LIN {X 0,Y 508.464,Z 856.949,A -85,B 0,C 180,E1 23996.123,E2 23996.123} C_VEL
LIN {X 0,Y 510.353,Z 835.895,A -85,B 0,C 180,E1 23994.699,E2 23994.699} C_VEL
LIN {X 0,Y 512.126,Z 815.37,A -85,B 0,C 180,E1 23993.529,E2 23993.529} C_VEL
LIN {X 0,Y 513.642,Z 794.189,A -85,B 0,C 180,E1 23992.545,E2 23992.545} C_VEL
LIN {X 0,Y 515.036,Z 772.161,A -85,B 0,C 180,E1 23991.717,E2 23991.717} C_VEL
LIN {X 0,Y 516.1,Z 749.861,A -85,B 0,C 180,E1 23991.103,E2 23991.103} C_VEL
LIN {X 0,Y 516.88,Z 725.33,A -85,B 0,C 180,E1 23990.627,E2 23990.627} C_VEL
LIN {X 0,Y 520.489,Z 517.525,A -85,B 0,C 180,E1 23987.247,E2 23987.247} C_VEL
LIN {X 0,Y 522.256,Z 415.583,A -85,B 0,C 180,E1 23985.539,E2 23985.539} C_VEL
LIN {X 0,Y 521.351,Z 412.142,A -85,B 0,C 180,E1 23985.377,E2 23985.377} C_VEL
LIN {X 0,Y 506.153,Z 388.849,A -85,B 0,C 180,E1 23983.194,E2 23983.194} C_VEL
LIN {X 0,Y 500.353,Z 377.109,A -85,B 0,C 180,E1 23981.409,E2 23981.409} C_VEL
LIN {X 0,Y 498.571,Z 373.357,A -85,B 0,C 180,E1 23980.826,E2 23980.826} C_VEL
LIN {X 0,Y 496.991,Z 370.279,A -85,B 0,C 180,E1 23980.325,E2 23980.325} C_VEL
LIN {X 0,Y 496.775,Z 369.171,A -85,B 0,C 180,E1 23980.17,E2 23980.17} C_VEL
LIN {X 0,Y 496.727,Z 369.173,A -85,B 0,C 180,E1 23976.714,E2 23976.714} C_VEL
LIN {X 0,Y 496.716,Z 369.158,A -85,B 0,C 180,E1 23973.146,E2 23973.146} C_VEL
LIN {X 0,Y 496.773,Z 369.141,A -85,B 0,C 180,E1 23969.81,E2 23969.81} C_VEL
LIN {X 0,Y 496.717,Z 369.17,A -85,B 0,C 180,E1 23966.409,E2 23966.409} C_VEL
LIN {X 0,Y 496.704,Z 369.151,A -85,B 0,C 180,E1 23962.861,E2 23962.861} C_VEL
LIN {X 0,Y 496.76,Z 369.159,A -85,B 0,C 180,E1 23959.519,E2 23959.519} C_VEL
LIN {X 0,Y 496.704,Z 369.158,A -85,B 0,C 180,E1 23956.128,E2 23956.128} C_VEL
LIN {X 0,Y 496.693,Z 369.168,A -85,B 0,C 180,E1 23952.556,E2 23952.556} C_VEL
LIN {X 0,Y 496.742,Z 369.166,A -85,B 0,C 180,E1 23949.149,E2 23949.149} C_VEL
LIN {X 0,Y 496.691,Z 369.172,A -85,B 0,C 180,E1 23945.892,E2 23945.892} C_VEL
LIN {X 0,Y 496.69,Z 369.167,A -85,B 0,C 180,E1 23942.307,E2 23942.307} C_VEL
LIN {X 0,Y 496.758,Z 369.164,A -85,B 0,C 180,E1 23938.962,E2 23938.962} C_VEL
LIN {X 0,Y 496.711,Z 369.174,A -85,B 0,C 180,E1 23935.497,E2 23935.497} C_VEL
LIN {X 0,Y 496.703,Z 369.171,A -85,B 0,C 180,E1 23932.002,E2 23932.002} C_VEL
LIN {X 0,Y 496.76,Z 369.165,A -85,B 0,C 180,E1 23928.624,E2 23928.624} C_VEL
LIN {X 0,Y 496.725,Z 369.174,A -85,B 0,C 180,E1 23925.188,E2 23925.188} C_VEL
LIN {X 0,Y 496.712,Z 369.149,A -85,B 0,C 180,E1 23921.698,E2 23921.698} C_VEL
LIN {X 0,Y 496.768,Z 369.16,A -85,B 0,C 180,E1 23918.263,E2 23918.263} C_VEL
LIN {X 0,Y 496.746,Z 369.154,A -85,B 0,C 180,E1 23914.74,E2 23914.74} C_VEL
LIN {X 0,Y 496.721,Z 369.154,A -85,B 0,C 180,E1 23911.243,E2 23911.243} C_VEL
LIN {X 0,Y 496.754,Z 369.169,A -85,B 0,C 180,E1 23907.765,E2 23907.765} C_VEL
LIN {X 0,Y 496.766,Z 369.148,A -85,B 0,C 180,E1 23904.289,E2 23904.289} C_VEL
LIN {X 0,Y 496.733,Z 369.148,A -85,B 0,C 180,E1 23900.792,E2 23900.792} C_VEL
LIN {X 0,Y 496.803,Z 369.408,A -85,B 0,C 180,E1 23897.786,E2 23897.786} C_VEL
LIN {X 0,Y 498.038,Z 372.602,A -85,B 0,C 180,E1 23897.561,E2 23897.561} C_VEL
LIN {X 0,Y 500.713,Z 375.613,A -85,B 0,C 180,E1 23897.161,E2 23897.161} C_VEL
LIN {X 0,Y 503.415,Z 379.529,A -85,B 0,C 180,E1 23896.747,E2 23896.747} C_VEL
LIN {X 0,Y 505.239,Z 382.053,A -85,B 0,C 180,E1 23896.474,E2 23896.474} C_VEL
LIN {X 0,Y 515.597,Z 396.493,A -85,B 0,C 180,E1 23894.982,E2 23894.982} C_VEL
LIN {X 0,Y 522.157,Z 406.331,A -85,B 0,C 180,E1 23894.073,E2 23894.073} C_VEL
LIN {X 0,Y 521.852,Z 421.709,A -85,B 0,C 180,E1 23893.817,E2 23893.817} C_VEL
LIN {X 0,Y 520.999,Z 429.411,A -85,B 0,C 180,E1 23893.763,E2 23893.763} C_VEL
LIN {X 0,Y 516.075,Z 450.049,A -85,B 0,C 180,E1 23893.901,E2 23893.901} C_VEL
LIN {X 0,Y 515.405,Z 456.658,A -85,B 0,C 180,E1 23893.847,E2 23893.847} C_VEL
LIN {X 0,Y 511.252,Z 667.268,A -85,B 0,C 180,E1 23890.36,E2 23890.36} C_VEL
LIN {X 0,Y 510.217,Z 713.646,A -85,B 0,C 180,E1 23889.568,E2 23889.568} C_VEL
LIN {X 0,Y 509.142,Z 735.14,A -85,B 0,C 180,E1 23889.014,E2 23889.014} C_VEL
LIN {X 0,Y 507.831,Z 756.494,A -85,B 0,C 180,E1 23888.289,E2 23888.289} C_VEL
LIN {X 0,Y 506.068,Z 778.939,A -85,B 0,C 180,E1 23887.296,E2 23887.296} C_VEL
LIN {X 0,Y 504.16,Z 801.229,A -85,B 0,C 180,E1 23886.082,E2 23886.082} C_VEL
LIN {X 0,Y 502.303,Z 820.309,A -85,B 0,C 180,E1 23884.835,E2 23884.835} C_VEL
LIN {X 0,Y 500.115,Z 841.41,A -85,B 0,C 180,E1 23883.211,E2 23883.211} C_VEL
LIN {X 0,Y 498.19,Z 859.526,A -85,B 0,C 180,E1 23881.585,E2 23881.585} C_VEL
LIN {X 0,Y 496.137,Z 878.107,A -85,B 0,C 180,E1 23879.649,E2 23879.649} C_VEL
LIN {X 0,Y 494.326,Z 895.329,A -85,B 0,C 180,E1 23877.589,E2 23877.589} C_VEL
LIN {X 0,Y 492.667,Z 911.402,A -85,B 0,C 180,E1 23875.351,E2 23875.351} C_VEL
LIN {X 0,Y 491.199,Z 926.819,A -85,B 0,C 180,E1 23872.876,E2 23872.876} C_VEL
LIN {X 0,Y 490.091,Z 940.046,A -85,B 0,C 180,E1 23870.415,E2 23870.415} C_VEL
LIN {X 0,Y 489.24,Z 951.697,A -85,B 0,C 180,E1 23867.849,E2 23867.849} C_VEL
LIN {X 0,Y 488.644,Z 961.975,A -85,B 0,C 180,E1 23865.181,E2 23865.181} C_VEL
LIN {X 0,Y 488.286,Z 969.634,A -85,B 0,C 180,E1 23862.775,E2 23862.775} C_VEL
LIN {X 0,Y 488.034,Z 976.716,A -85,B 0,C 180,E1 23860.027,E2 23860.027} C_VEL
LIN {X 0,Y 487.954,Z 981.385,A -85,B 0,C 180,E1 23857.653,E2 23857.653} C_VEL
LIN {X 0,Y 487.914,Z 985.231,A -85,B 0,C 180,E1 23854.937,E2 23854.937} C_VEL
LIN {X 0,Y 487.909,Z 987.232,A -85,B 0,C 180,E1 23852.466,E2 23852.466} C_VEL
LIN {X 0,Y 487.908,Z 987.992,A -85,B 0,C 180,E1 23849.882,E2 23849.882} C_VEL
LIN {X 0,Y 487.904,Z 987.148,A -85,B 0,C 180,E1 23847.298,E2 23847.298} C_VEL
LIN {X 0,Y 487.918,Z 984.97,A -85,B 0,C 180,E1 23844.709,E2 23844.709} C_VEL
LIN {X 0,Y 487.969,Z 981.128,A -85,B 0,C 180,E1 23842.11,E2 23842.11} C_VEL
LIN {X 0,Y 488.079,Z 975.882,A -85,B 0,C 180,E1 23839.496,E2 23839.496} C_VEL
LIN {X 0,Y 488.32,Z 968.838,A -85,B 0,C 180,E1 23836.864,E2 23836.864} C_VEL
LIN {X 0,Y 488.735,Z 960.16,A -85,B 0,C 180,E1 23834.213,E2 23834.213} C_VEL
LIN {X 0,Y 489.315,Z 950.523,A -85,B 0,C 180,E1 23831.784,E2 23831.784} C_VEL
LIN {X 0,Y 490.256,Z 937.895,A -85,B 0,C 180,E1 23829.079,E2 23829.079} C_VEL
LIN {X 0,Y 491.348,Z 925.2,A -85,B 0,C 180,E1 23826.75,E2 23826.75} C_VEL
LIN {X 0,Y 492.769,Z 910.298,A -85,B 0,C 180,E1 23824.396,E2 23824.396} C_VEL
LIN {X 0,Y 494.415,Z 894.536,A -85,B 0,C 180,E1 23822.219,E2 23822.219} C_VEL
LIN {X 0,Y 496.191,Z 877.593,A -85,B 0,C 180,E1 23820.203,E2 23820.203} C_VEL
LIN {X 0,Y 498.305,Z 858.41,A -85,B 0,C 180,E1 23818.22,E2 23818.22} C_VEL
LIN {X 0,Y 500.249,Z 840.17,A -85,B 0,C 180,E1 23816.593,E2 23816.593} C_VEL
LIN {X 0,Y 502.368,Z 819.664,A -85,B 0,C 180,E1 23815.03,E2 23815.03} C_VEL
LIN {X 0,Y 504.234,Z 800.49,A -85,B 0,C 180,E1 23813.783,E2 23813.783} C_VEL
LIN {X 0,Y 506.062,Z 779,A -85,B 0,C 180,E1 23812.617,E2 23812.617} C_VEL
LIN {X 0,Y 507.824,Z 756.603,A -85,B 0,C 180,E1 23811.625,E2 23811.625} C_VEL
LIN {X 0,Y 509.13,Z 735.348,A -85,B 0,C 180,E1 23810.903,E2 23810.903} C_VEL
LIN {X 0,Y 510.191,Z 714.187,A -85,B 0,C 180,E1 23810.354,E2 23810.354} C_VEL
LIN {X 0,Y 511.145,Z 673.08,A -85,B 0,C 180,E1 23809.645,E2 23809.645} C_VEL
LIN {X 0,Y 515.353,Z 459.338,A -85,B 0,C 180,E1 23806.108,E2 23806.108} C_VEL
LIN {X 0,Y 516.278,Z 409.582,A -85,B 0,C 180,E1 23805.257,E2 23805.257} C_VEL
LIN {X 0,Y 502.991,Z 390.592,A -85,B 0,C 180,E1 23803.338,E2 23803.338} C_VEL
LIN {X 0,Y 498.896,Z 385.123,A -85,B 0,C 180,E1 23802.719,E2 23802.719} C_VEL
LIN {X 0,Y 495.764,Z 380.744,A -85,B 0,C 180,E1 23802.23,E2 23802.23} C_VEL
LIN {X 0,Y 493.031,Z 376.923,A -85,B 0,C 180,E1 23801.793,E2 23801.793} C_VEL
LIN {X 0,Y 492.228,Z 375.754,A -85,B 0,C 180,E1 23801.663,E2 23801.663} C_VEL
LIN {X 0,Y 489.757,Z 373.065,A -85,B 0,C 180,E1 23801.275,E2 23801.275} C_VEL
LIN {X 0,Y 488.804,Z 370.162,A -85,B 0,C 180,E1 23801.073,E2 23801.073} C_VEL
LIN {X 0,Y 488.818,Z 370.152,A -85,B 0,C 180,E1 23797.481,E2 23797.481} C_VEL
LIN {X 0,Y 488.831,Z 370.129,A -85,B 0,C 180,E1 23793.866,E2 23793.866} C_VEL
LIN {X 0,Y 488.803,Z 370.14,A -85,B 0,C 180,E1 23790.332,E2 23790.332} C_VEL
LIN {X 0,Y 488.79,Z 370.162,A -85,B 0,C 180,E1 23786.746,E2 23786.746} C_VEL
LIN {X 0,Y 488.816,Z 370.127,A -85,B 0,C 180,E1 23783.252,E2 23783.252} C_VEL
LIN {X 0,Y 488.82,Z 370.159,A -85,B 0,C 180,E1 23779.725,E2 23779.725} C_VEL
LIN {X 0,Y 488.773,Z 370.134,A -85,B 0,C 180,E1 23776.276,E2 23776.276} C_VEL
LIN {X 0,Y 488.791,Z 370.156,A -85,B 0,C 180,E1 23772.763,E2 23772.763} C_VEL
LIN {X 0,Y 488.823,Z 370.157,A -85,B 0,C 180,E1 23769.299,E2 23769.299} C_VEL
LIN {X 0,Y 488.768,Z 370.161,A -85,B 0,C 180,E1 23765.871,E2 23765.871} C_VEL
LIN {X 0,Y 488.764,Z 370.161,A -85,B 0,C 180,E1 23762.228,E2 23762.228} C_VEL
LIN {X 0,Y 488.817,Z 370.159,A -85,B 0,C 180,E1 23758.828,E2 23758.828} C_VEL
LIN {X 0,Y 488.771,Z 370.163,A -85,B 0,C 180,E1 23755.307,E2 23755.307} C_VEL
LIN {X 0,Y 488.748,Z 370.163,A -85,B 0,C 180,E1 23751.885,E2 23751.885} C_VEL
LIN {X 0,Y 488.798,Z 370.16,A -85,B 0,C 180,E1 23748.436,E2 23748.436} C_VEL
LIN {X 0,Y 488.77,Z 370.165,A -85,B 0,C 180,E1 23745.064,E2 23745.064} C_VEL
LIN {X 0,Y 488.757,Z 370.14,A -85,B 0,C 180,E1 23741.514,E2 23741.514} C_VEL
LIN {X 0,Y 488.796,Z 370.152,A -85,B 0,C 180,E1 23738.017,E2 23738.017} C_VEL
LIN {X 0,Y 488.802,Z 370.15,A -85,B 0,C 180,E1 23734.561,E2 23734.561} C_VEL
LIN {X 0,Y 488.768,Z 370.137,A -85,B 0,C 180,E1 23731.098,E2 23731.098} C_VEL
LIN {X 0,Y 488.795,Z 370.155,A -85,B 0,C 180,E1 23727.593,E2 23727.593} C_VEL
LIN {X 0,Y 488.829,Z 370.157,A -85,B 0,C 180,E1 23724.054,E2 23724.054} C_VEL
LIN {X 0,Y 488.799,Z 370.271,A -85,B 0,C 180,E1 23720.776,E2 23720.776} C_VEL
LIN {X 0,Y 490.062,Z 373.556,A -85,B 0,C 180,E1 23720.273,E2 23720.273} C_VEL
LIN {X 0,Y 491.239,Z 375.449,A -85,B 0,C 180,E1 23719.927,E2 23719.927} C_VEL
LIN {X 0,Y 497.884,Z 388.868,A -85,B 0,C 180,E1 23717.812,E2 23717.812} C_VEL
LIN {X 0,Y 511.426,Z 409.267,A -85,B 0,C 180,E1 23715.777,E2 23715.777} C_VEL
LIN {X 0,Y 516.558,Z 417.775,A -85,B 0,C 180,E1 23715.037,E2 23715.037} C_VEL
LIN {X 0,Y 513.166,Z 591.207,A -85,B 0,C 180,E1 23712.135,E2 23712.135} C_VEL
LIN {X 0,Y 510.26,Z 740.048,A -85,B 0,C 180,E1 23709.677,E2 23709.677} C_VEL
LIN {X 0,Y 509.209,Z 762.982,A -85,B 0,C 180,E1 23709.115,E2 23709.115} C_VEL
LIN {X 0,Y 508.022,Z 782.983,A -85,B 0,C 180,E1 23708.457,E2 23708.457} C_VEL
LIN {X 0,Y 506.378,Z 805.177,A -85,B 0,C 180,E1 23707.523,E2 23707.523} C_VEL
LIN {X 0,Y 504.581,Z 826.539,A -85,B 0,C 180,E1 23706.407,E2 23706.407} C_VEL
LIN {X 0,Y 502.609,Z 847.281,A -85,B 0,C 180,E1 23705.09,E2 23705.09} C_VEL
LIN {X 0,Y 500.556,Z 867.467,A -85,B 0,C 180,E1 23703.59,E2 23703.59} C_VEL
LIN {X 0,Y 498.488,Z 886.631,A -85,B 0,C 180,E1 23701.902,E2 23701.902} C_VEL
LIN {X 0,Y 496.409,Z 905.703,A -85,B 0,C 180,E1 23699.965,E2 23699.965} C_VEL
LIN {X 0,Y 494.669,Z 921.952,A -85,B 0,C 180,E1 23698.055,E2 23698.055} C_VEL
LIN {X 0,Y 492.895,Z 938.97,A -85,B 0,C 180,E1 23695.754,E2 23695.754} C_VEL
LIN {X 0,Y 491.484,Z 953.859,A -85,B 0,C 180,E1 23693.438,E2 23693.438} C_VEL
LIN {X 0,Y 490.319,Z 967.096,A -85,B 0,C 180,E1 23691.03,E2 23691.03} C_VEL
LIN {X 0,Y 489.404,Z 979.297,A -85,B 0,C 180,E1 23688.46,E2 23688.46} C_VEL
LIN {X 0,Y 488.783,Z 989.073,A -85,B 0,C 180,E1 23686.029,E2 23686.029} C_VEL
LIN {X 0,Y 488.338,Z 998.352,A -85,B 0,C 180,E1 23683.256,E2 23683.256} C_VEL
LIN {X 0,Y 488.1,Z 1004.868,A -85,B 0,C 180,E1 23680.862,E2 23680.862} C_VEL
LIN {X 0,Y 487.978,Z 1010.636,A -85,B 0,C 180,E1 23678.127,E2 23678.127} C_VEL
LIN {X 0,Y 487.913,Z 1014.438,A -85,B 0,C 180,E1 23675.645,E2 23675.645} C_VEL
LIN {X 0,Y 487.89,Z 1016.986,A -85,B 0,C 180,E1 23672.937,E2 23672.937} C_VEL
LIN {X 0,Y 487.885,Z 1017.895,A -85,B 0,C 180,E1 23670.587,E2 23670.587} C_VEL
LIN {X 0,Y 487.914,Z 1017.393,A -85,B 0,C 180,E1 23667.769,E2 23667.769} C_VEL
LIN {X 0,Y 487.906,Z 1015.502,A -85,B 0,C 180,E1 23665.299,E2 23665.299} C_VEL
LIN {X 0,Y 487.933,Z 1011.876,A -85,B 0,C 180,E1 23662.584,E2 23662.584} C_VEL
LIN {X 0,Y 488.017,Z 1007.347,A -85,B 0,C 180,E1 23660.222,E2 23660.222} C_VEL
LIN {X 0,Y 488.242,Z 1000.825,A -85,B 0,C 180,E1 23657.585,E2 23657.585} C_VEL
LIN {X 0,Y 488.592,Z 992.944,A -85,B 0,C 180,E1 23655.06,E2 23655.06} C_VEL
LIN {X 0,Y 489.199,Z 982.338,A -85,B 0,C 180,E1 23652.257,E2 23652.257} C_VEL
LIN {X 0,Y 489.978,Z 971.429,A -85,B 0,C 180,E1 23649.829,E2 23649.829} C_VEL
LIN {X 0,Y 491.056,Z 958.469,A -85,B 0,C 180,E1 23647.37,E2 23647.37} C_VEL
LIN {X 0,Y 492.405,Z 944.233,A -85,B 0,C 180,E1 23645.02,E2 23645.02} C_VEL
LIN {X 0,Y 493.963,Z 928.434,A -85,B 0,C 180,E1 23642.78,E2 23642.78} C_VEL
LIN {X 0,Y 495.925,Z 910.148,A -85,B 0,C 180,E1 23640.536,E2 23640.536} C_VEL
LIN {X 0,Y 497.859,Z 892.56,A -85,B 0,C 180,E1 23638.662,E2 23638.662} C_VEL
LIN {X 0,Y 499.911,Z 873.362,A -85,B 0,C 180,E1 23636.91,E2 23636.91} C_VEL
LIN {X 0,Y 501.985,Z 853.573,A -85,B 0,C 180,E1 23635.347,E2 23635.347} C_VEL
LIN {X 0,Y 503.895,Z 833.882,A -85,B 0,C 180,E1 23634.037,E2 23634.037} C_VEL
LIN {X 0,Y 505.798,Z 812.769,A -85,B 0,C 180,E1 23632.848,E2 23632.848} C_VEL
LIN {X 0,Y 507.33,Z 792.54,A -85,B 0,C 180,E1 23631.918,E2 23631.918} C_VEL
LIN {X 0,Y 508.864,Z 769.286,A -85,B 0,C 180,E1 23631.071,E2 23631.071} C_VEL
LIN {X 0,Y 509.898,Z 748.81,A -85,B 0,C 180,E1 23630.516,E2 23630.516} C_VEL
LIN {X 0,Y 510.736,Z 722.059,A -85,B 0,C 180,E1 23630.006,E2 23630.006} C_VEL
LIN {X 0,Y 514.648,Z 514.981,A -85,B 0,C 180,E1 23626.601,E2 23626.601} C_VEL
LIN {X 0,Y 516.488,Z 417.402,A -85,B 0,C 180,E1 23624.948,E2 23624.948} C_VEL
LIN {X 0,Y 502.74,Z 395.952,A -85,B 0,C 180,E1 23622.935,E2 23622.935} C_VEL
LIN {X 0,Y 497.647,Z 388.466,A -85,B 0,C 180,E1 23622.149,E2 23622.149} C_VEL
LIN {X 0,Y 492.504,Z 378.211,A -85,B 0,C 180,E1 23620.515,E2 23620.515} C_VEL
LIN {X 0,Y 490.79,Z 374.486,A -85,B 0,C 180,E1 23619.921,E2 23619.921} C_VEL
LIN {X 0,Y 488.97,Z 371.128,A -85,B 0,C 180,E1 23619.338,E2 23619.338} C_VEL
LIN {X 0,Y 488.783,Z 370.16,A -85,B 0,C 180,E1 23619.178,E2 23619.178} C_VEL
LIN {X 0,Y 488.811,Z 370.153,A -85,B 0,C 180,E1 23615.659,E2 23615.659} C_VEL
LIN {X 0,Y 488.82,Z 370.155,A -85,B 0,C 180,E1 23612.128,E2 23612.128} C_VEL
LIN {X 0,Y 488.769,Z 370.135,A -85,B 0,C 180,E1 23608.733,E2 23608.733} C_VEL
LIN {X 0,Y 488.783,Z 370.145,A -85,B 0,C 180,E1 23605.181,E2 23605.181} C_VEL
LIN {X 0,Y 488.825,Z 370.146,A -85,B 0,C 180,E1 23601.729,E2 23601.729} C_VEL
LIN {X 0,Y 488.763,Z 370.135,A -85,B 0,C 180,E1 23598.239,E2 23598.239} C_VEL
LIN {X 0,Y 488.758,Z 370.164,A -85,B 0,C 180,E1 23594.647,E2 23594.647} C_VEL
LIN {X 0,Y 488.806,Z 370.162,A -85,B 0,C 180,E1 23591.205,E2 23591.205} C_VEL
LIN {X 0,Y 488.766,Z 370.162,A -85,B 0,C 180,E1 23587.759,E2 23587.759} C_VEL
LIN {X 0,Y 488.748,Z 370.164,A -85,B 0,C 180,E1 23584.223,E2 23584.223} C_VEL
LIN {X 0,Y 488.796,Z 370.162,A -85,B 0,C 180,E1 23580.82,E2 23580.82} C_VEL
LIN {X 0,Y 488.778,Z 370.157,A -85,B 0,C 180,E1 23577.42,E2 23577.42} C_VEL
LIN {X 0,Y 488.759,Z 370.16,A -85,B 0,C 180,E1 23573.893,E2 23573.893} C_VEL
LIN {X 0,Y 488.8,Z 370.158,A -85,B 0,C 180,E1 23570.463,E2 23570.463} C_VEL
LIN {X 0,Y 488.804,Z 370.154,A -85,B 0,C 180,E1 23566.996,E2 23566.996} C_VEL
LIN {X 0,Y 488.77,Z 370.141,A -85,B 0,C 180,E1 23563.597,E2 23563.597} C_VEL
LIN {X 0,Y 488.807,Z 370.159,A -85,B 0,C 180,E1 23560.15,E2 23560.15} C_VEL
LIN {X 0,Y 488.816,Z 370.128,A -85,B 0,C 180,E1 23556.679,E2 23556.679} C_VEL
LIN {X 0,Y 488.786,Z 370.162,A -85,B 0,C 180,E1 23553.123,E2 23553.123} C_VEL
LIN {X 0,Y 488.793,Z 370.139,A -85,B 0,C 180,E1 23549.516,E2 23549.516} C_VEL
LIN {X 0,Y 488.831,Z 370.133,A -85,B 0,C 180,E1 23546.055,E2 23546.055} C_VEL
LIN {X 0,Y 488.818,Z 370.155,A -85,B 0,C 180,E1 23542.443,E2 23542.443} C_VEL
LIN {X 0,Y 488.797,Z 370.162,A -85,B 0,C 180,E1 23538.896,E2 23538.896} C_VEL
LIN {X 0,Y 488.832,Z 370.403,A -85,B 0,C 180,E1 23538.816,E2 23538.816} C_VEL
LIN {X 0,Y 490.061,Z 373.569,A -85,B 0,C 180,E1 23538.581,E2 23538.581} C_VEL
LIN {X 0,Y 492.913,Z 376.68,A -85,B 0,C 180,E1 23538.136,E2 23538.136} C_VEL
LIN {X 0,Y 495.559,Z 380.548,A -85,B 0,C 180,E1 23537.71,E2 23537.71} C_VEL
LIN {X 0,Y 497.277,Z 382.868,A -85,B 0,C 180,E1 23537.442,E2 23537.442} C_VEL
LIN {X 0,Y 504.541,Z 392.801,A -85,B 0,C 180,E1 23536.339,E2 23536.339} C_VEL
LIN {X 0,Y 516.37,Z 409.728,A -85,B 0,C 180,E1 23534.64,E2 23534.64} C_VEL
LIN {X 0,Y 515.405,Z 456.658,A -85,B 0,C 180,E1 23533.847,E2 23533.847} C_VEL
LIN {X 0,Y 514.529,Z 464.362,A -85,B 0,C 180,E1 23533.795,E2 23533.795} C_VEL
LIN {X 0,Y 509.557,Z 484.99,A -85,B 0,C 180,E1 23533.94,E2 23533.94} C_VEL
LIN {X 0,Y 508.893,Z 491.597,A -85,B 0,C 180,E1 23533.886,E2 23533.886} C_VEL
LIN {X 0,Y 504.452,Z 702.056,A -85,B 0,C 180,E1 23530.374,E2 23530.374} C_VEL
LIN {X 0,Y 503.552,Z 723.847,A -85,B 0,C 180,E1 23529.915,E2 23529.915} C_VEL
LIN {X 0,Y 502.14,Z 747.778,A -85,B 0,C 180,E1 23529.189,E2 23529.189} C_VEL
LIN {X 0,Y 500.66,Z 767.864,A -85,B 0,C 180,E1 23528.39,E2 23528.39} C_VEL
LIN {X 0,Y 498.747,Z 789.324,A -85,B 0,C 180,E1 23527.327,E2 23527.327} C_VEL
LIN {X 0,Y 496.745,Z 809.274,A -85,B 0,C 180,E1 23526.134,E2 23526.134} C_VEL
LIN {X 0,Y 494.552,Z 829.67,A -85,B 0,C 180,E1 23524.684,E2 23524.684} C_VEL
LIN {X 0,Y 492.413,Z 848.758,A -85,B 0,C 180,E1 23523.103,E2 23523.103} C_VEL
LIN {X 0,Y 490.161,Z 867.608,A -85,B 0,C 180,E1 23521.273,E2 23521.273} C_VEL
LIN {X 0,Y 488.127,Z 885.24,A -85,B 0,C 180,E1 23519.307,E2 23519.307} C_VEL
LIN {X 0,Y 486.237,Z 901.358,A -85,B 0,C 180,E1 23517.224,E2 23517.224} C_VEL
LIN {X 0,Y 484.434,Z 917.974,A -85,B 0,C 180,E1 23514.749,E2 23514.749} C_VEL
LIN {X 0,Y 483.042,Z 932.215,A -85,B 0,C 180,E1 23512.293,E2 23512.293} C_VEL
LIN {X 0,Y 481.928,Z 944.678,A -85,B 0,C 180,E1 23509.763,E2 23509.763} C_VEL
LIN {X 0,Y 481.074,Z 956.154,A -85,B 0,C 180,E1 23507.038,E2 23507.038} C_VEL
LIN {X 0,Y 480.559,Z 964.819,A -85,B 0,C 180,E1 23504.579,E2 23504.579} C_VEL
LIN {X 0,Y 480.195,Z 972.938,A -85,B 0,C 180,E1 23501.772,E2 23501.772} C_VEL
LIN {X 0,Y 480.019,Z 978.499,A -85,B 0,C 180,E1 23499.349,E2 23499.349} C_VEL
LIN {X 0,Y 479.936,Z 983.262,A -85,B 0,C 180,E1 23496.578,E2 23496.578} C_VEL
LIN {X 0,Y 479.913,Z 986.027,A -85,B 0,C 180,E1 23494.181,E2 23494.181} C_VEL
LIN {X 0,Y 479.908,Z 987.75,A -85,B 0,C 180,E1 23491.313,E2 23491.313} C_VEL
LIN {X 0,Y 479.892,Z 987.813,A -85,B 0,C 180,E1 23488.925,E2 23488.925} C_VEL
LIN {X 0,Y 479.899,Z 986.563,A -85,B 0,C 180,E1 23486.297,E2 23486.297} C_VEL
LIN {X 0,Y 479.934,Z 983.86,A -85,B 0,C 180,E1 23483.781,E2 23483.781} C_VEL
LIN {X 0,Y 480.003,Z 979.68,A -85,B 0,C 180,E1 23481.134,E2 23481.134} C_VEL
LIN {X 0,Y 480.148,Z 973.768,A -85,B 0,C 180,E1 23478.469,E2 23478.469} C_VEL
LIN {X 0,Y 480.462,Z 966.602,A -85,B 0,C 180,E1 23475.875,E2 23475.875} C_VEL
LIN {X 0,Y 480.95,Z 957.861,A -85,B 0,C 180,E1 23473.33,E2 23473.33} C_VEL
LIN {X 0,Y 481.708,Z 947.373,A -85,B 0,C 180,E1 23470.731,E2 23470.731} C_VEL
LIN {X 0,Y 482.711,Z 935.413,A -85,B 0,C 180,E1 23468.239,E2 23468.239} C_VEL
LIN {X 0,Y 484.15,Z 920.709,A -85,B 0,C 180,E1 23465.607,E2 23465.607} C_VEL
LIN {X 0,Y 485.736,Z 906.057,A -85,B 0,C 180,E1 23463.34,E2 23463.34} C_VEL
LIN {X 0,Y 487.531,Z 889.966,A -85,B 0,C 180,E1 23461.19,E2 23461.19} C_VEL
LIN {X 0,Y 489.606,Z 872.681,A -85,B 0,C 180,E1 23459.167,E2 23459.167} C_VEL
LIN {X 0,Y 491.702,Z 854.474,A -85,B 0,C 180,E1 23457.337,E2 23457.337} C_VEL
LIN {X 0,Y 494.091,Z 833.949,A -85,B 0,C 180,E1 23455.56,E2 23455.56} C_VEL
LIN {X 0,Y 496.132,Z 815.146,A -85,B 0,C 180,E1 23454.17,E2 23454.17} C_VEL
LIN {X 0,Y 498.35,Z 793.207,A -85,B 0,C 180,E1 23452.799,E2 23452.799} C_VEL
LIN {X 0,Y 500.3,Z 772.386,A -85,B 0,C 180,E1 23451.722,E2 23451.722} C_VEL
LIN {X 0,Y 501.962,Z 750.45,A -85,B 0,C 180,E1 23450.819,E2 23450.819} C_VEL
LIN {X 0,Y 503.317,Z 729.014,A -85,B 0,C 180,E1 23450.127,E2 23450.127} C_VEL
LIN {X 0,Y 504.316,Z 705.93,A -85,B 0,C 180,E1 23449.607,E2 23449.607} C_VEL
LIN {X 0,Y 508.655,Z 502.265,A -85,B 0,C 180,E1 23446.204,E2 23446.204} C_VEL
LIN {X 0,Y 510.494,Z 413.361,A -85,B 0,C 180,E1 23444.68,E2 23444.68} C_VEL
LIN {X 0,Y 498.725,Z 396.42,A -85,B 0,C 180,E1 23442.933,E2 23442.933} C_VEL
LIN {X 0,Y 491.408,Z 386.502,A -85,B 0,C 180,E1 23441.787,E2 23441.787} C_VEL
LIN {X 0,Y 488.039,Z 381.9,A -85,B 0,C 180,E1 23441.237,E2 23441.237} C_VEL
LIN {X 0,Y 485.212,Z 378.061,A -85,B 0,C 180,E1 23440.766,E2 23440.766} C_VEL
LIN {X 0,Y 484.28,Z 376.743,A -85,B 0,C 180,E1 23440.608,E2 23440.608} C_VEL
LIN {X 0,Y 481.8,Z 373.956,A -85,B 0,C 180,E1 23440.196,E2 23440.196} C_VEL
LIN {X 0,Y 480.89,Z 371.123,A -85,B 0,C 180,E1 23439.976,E2 23439.976} C_VEL
LIN {X 0,Y 480.879,Z 371.144,A -85,B 0,C 180,E1 23436.341,E2 23436.341} C_VEL
LIN {X 0,Y 480.856,Z 371.146,A -85,B 0,C 180,E1 23432.726,E2 23432.726} C_VEL
LIN {X 0,Y 480.86,Z 371.118,A -85,B 0,C 180,E1 23429.115,E2 23429.115} C_VEL
LIN {X 0,Y 480.893,Z 371.138,A -85,B 0,C 180,E1 23425.543,E2 23425.543} C_VEL
LIN {X 0,Y 480.864,Z 371.133,A -85,B 0,C 180,E1 23421.98,E2 23421.98} C_VEL
LIN {X 0,Y 480.839,Z 371.132,A -85,B 0,C 180,E1 23418.426,E2 23418.426} C_VEL
LIN {X 0,Y 480.864,Z 371.138,A -85,B 0,C 180,E1 23414.942,E2 23414.942} C_VEL
LIN {X 0,Y 480.882,Z 371.139,A -85,B 0,C 180,E1 23411.393,E2 23411.393} C_VEL
LIN {X 0,Y 480.832,Z 371.143,A -85,B 0,C 180,E1 23407.889,E2 23407.889} C_VEL
LIN {X 0,Y 480.828,Z 371.147,A -85,B 0,C 180,E1 23404.293,E2 23404.293} C_VEL
LIN {X 0,Y 480.877,Z 371.14,A -85,B 0,C 180,E1 23400.834,E2 23400.834} C_VEL
LIN {X 0,Y 480.832,Z 371.143,A -85,B 0,C 180,E1 23397.378,E2 23397.378} C_VEL
LIN {X 0,Y 480.811,Z 371.144,A -85,B 0,C 180,E1 23393.912,E2 23393.912} C_VEL
LIN {X 0,Y 480.86,Z 371.142,A -85,B 0,C 180,E1 23390.546,E2 23390.546} C_VEL
LIN {X 0,Y 480.826,Z 371.146,A -85,B 0,C 180,E1 23387.144,E2 23387.144} C_VEL
LIN {X 0,Y 480.818,Z 371.141,A -85,B 0,C 180,E1 23383.696,E2 23383.696} C_VEL
LIN {X 0,Y 480.865,Z 371.143,A -85,B 0,C 180,E1 23380.189,E2 23380.189} C_VEL
LIN {X 0,Y 480.851,Z 371.122,A -85,B 0,C 180,E1 23376.73,E2 23376.73} C_VEL
LIN {X 0,Y 480.831,Z 371.153,A -85,B 0,C 180,E1 23373.177,E2 23373.177} C_VEL
LIN {X 0,Y 480.852,Z 371.133,A -85,B 0,C 180,E1 23369.636,E2 23369.636} C_VEL
LIN {X 0,Y 480.888,Z 371.118,A -85,B 0,C 180,E1 23366.136,E2 23366.136} C_VEL
LIN {X 0,Y 480.85,Z 371.131,A -85,B 0,C 180,E1 23362.582,E2 23362.582} C_VEL
LIN {X 0,Y 480.902,Z 371.209,A -85,B 0,C 180,E1 23361.797,E2 23361.797} C_VEL
LIN {X 0,Y 481.869,Z 374.143,A -85,B 0,C 180,E1 23361.35,E2 23361.35} C_VEL
LIN {X 0,Y 483.362,Z 376.618,A -85,B 0,C 180,E1 23360.883,E2 23360.883} C_VEL
LIN {X 0,Y 488.149,Z 386.216,A -85,B 0,C 180,E1 23359.268,E2 23359.268} C_VEL
LIN {X 0,Y 489.762,Z 388.875,A -85,B 0,C 180,E1 23358.862,E2 23358.862} C_VEL
LIN {X 0,Y 502.739,Z 408.402,A -85,B 0,C 180,E1 23356.812,E2 23356.812} C_VEL
LIN {X 0,Y 510.89,Z 421.38,A -85,B 0,C 180,E1 23355.6,E2 23355.6} C_VEL
LIN {X 0,Y 506.323,Z 634.936,A -85,B 0,C 180,E1 23352.013,E2 23352.013} C_VEL
LIN {X 0,Y 504.072,Z 740.195,A -85,B 0,C 180,E1 23350.253,E2 23350.253} C_VEL
LIN {X 0,Y 502.943,Z 762.907,A -85,B 0,C 180,E1 23349.69,E2 23349.69} C_VEL
LIN {X 0,Y 501.64,Z 783.377,A -85,B 0,C 180,E1 23349.009,E2 23349.009} C_VEL
LIN {X 0,Y 499.815,Z 806.231,A -85,B 0,C 180,E1 23348.03,E2 23348.03} C_VEL
LIN {X 0,Y 497.913,Z 827.719,A -85,B 0,C 180,E1 23346.895,E2 23346.895} C_VEL
LIN {X 0,Y 495.813,Z 848.178,A -85,B 0,C 180,E1 23345.572,E2 23345.572} C_VEL
LIN {X 0,Y 493.62,Z 868.173,A -85,B 0,C 180,E1 23344.06,E2 23344.06} C_VEL
LIN {X 0,Y 491.387,Z 887.296,A -85,B 0,C 180,E1 23342.35,E2 23342.35} C_VEL
LIN {X 0,Y 489.084,Z 906.811,A -85,B 0,C 180,E1 23340.325,E2 23340.325} C_VEL
LIN {X 0,Y 487.196,Z 923.174,A -85,B 0,C 180,E1 23338.363,E2 23338.363} C_VEL
LIN {X 0,Y 485.369,Z 939.156,A -85,B 0,C 180,E1 23336.155,E2 23336.155} C_VEL
LIN {X 0,Y 483.887,Z 953.521,A -85,B 0,C 180,E1 23333.888,E2 23333.888} C_VEL
LIN {X 0,Y 482.621,Z 966.459,A -85,B 0,C 180,E1 23331.51,E2 23331.51} C_VEL
LIN {X 0,Y 481.597,Z 978.777,A -85,B 0,C 180,E1 23328.896,E2 23328.896} C_VEL
LIN {X 0,Y 480.903,Z 988.613,A -85,B 0,C 180,E1 23326.423,E2 23326.423} C_VEL
LIN {X 0,Y 480.407,Z 997.641,A -85,B 0,C 180,E1 23323.724,E2 23323.724} C_VEL
LIN {X 0,Y 480.13,Z 1004.262,A -85,B 0,C 180,E1 23321.288,E2 23321.288} C_VEL
LIN {X 0,Y 479.994,Z 1010.223,A -85,B 0,C 180,E1 23318.504,E2 23318.504} C_VEL
LIN {X 0,Y 479.921,Z 1014.119,A -85,B 0,C 180,E1 23315.979,E2 23315.979} C_VEL
LIN {X 0,Y 479.885,Z 1016.85,A -85,B 0,C 180,E1 23313.225,E2 23313.225} C_VEL
LIN {X 0,Y 479.886,Z 1017.85,A -85,B 0,C 180,E1 23310.836,E2 23310.836} C_VEL
LIN {X 0,Y 479.907,Z 1017.658,A -85,B 0,C 180,E1 23308.21,E2 23308.21} C_VEL
LIN {X 0,Y 479.908,Z 1015.843,A -85,B 0,C 180,E1 23305.58,E2 23305.58} C_VEL
LIN {X 0,Y 479.923,Z 1012.682,A -85,B 0,C 180,E1 23302.941,E2 23302.941} C_VEL
LIN {X 0,Y 480.019,Z 1008.085,A -85,B 0,C 180,E1 23300.409,E2 23300.409} C_VEL
LIN {X 0,Y 480.217,Z 1002.44,A -85,B 0,C 180,E1 23297.984,E2 23297.984} C_VEL
LIN {X 0,Y 480.598,Z 994.158,A -85,B 0,C 180,E1 23295.175,E2 23295.175} C_VEL
LIN {X 0,Y 481.171,Z 984.93,A -85,B 0,C 180,E1 23292.591,E2 23292.591} C_VEL
LIN {X 0,Y 482.007,Z 973.736,A -85,B 0,C 180,E1 23289.988,E2 23289.988} C_VEL
LIN {X 0,Y 483.131,Z 961.269,A -85,B 0,C 180,E1 23287.492,E2 23287.492} C_VEL
LIN {X 0,Y 484.504,Z 947.364,A -85,B 0,C 180,E1 23285.106,E2 23285.106} C_VEL
LIN {X 0,Y 486.252,Z 931.21,A -85,B 0,C 180,E1 23282.711,E2 23282.711} C_VEL
LIN {X 0,Y 488.214,Z 914.562,A -85,B 0,C 180,E1 23280.564,E2 23280.564} C_VEL
LIN {X 0,Y 490.252,Z 896.816,A -85,B 0,C 180,E1 23278.599,E2 23278.599} C_VEL
LIN {X 0,Y 492.529,Z 877.683,A -85,B 0,C 180,E1 23276.759,E2 23276.759} C_VEL
LIN {X 0,Y 494.584,Z 859.377,A -85,B 0,C 180,E1 23275.248,E2 23275.248} C_VEL
LIN {X 0,Y 496.882,Z 837.897,A -85,B 0,C 180,E1 23273.734,E2 23273.734} C_VEL
LIN {X 0,Y 498.751,Z 818.62,A -85,B 0,C 180,E1 23272.601,E2 23272.601} C_VEL
LIN {X 0,Y 500.634,Z 796.527,A -85,B 0,C 180,E1 23271.526,E2 23271.526} C_VEL
LIN {X 0,Y 502.138,Z 775.614,A -85,B 0,C 180,E1 23270.71,E2 23270.71} C_VEL
LIN {X 0,Y 503.532,Z 751.794,A -85,B 0,C 180,E1 23270.01,E2 23270.01} C_VEL
LIN {X 0,Y 504.431,Z 729.338,A -85,B 0,C 180,E1 23269.546,E2 23269.546} C_VEL
LIN {X 0,Y 508.688,Z 521.006,A -85,B 0,C 180,E1 23266.084,E2 23266.084} C_VEL
LIN {X 0,Y 510.779,Z 420.993,A -85,B 0,C 180,E1 23264.379,E2 23264.379} C_VEL
LIN {X 0,Y 496.823,Z 399.314,A -85,B 0,C 180,E1 23262.274,E2 23262.274} C_VEL
LIN {X 0,Y 489.042,Z 387.922,A -85,B 0,C 180,E1 23261.017,E2 23261.017} C_VEL
LIN {X 0,Y 484.735,Z 379.412,A -85,B 0,C 180,E1 23259.596,E2 23259.596} C_VEL
LIN {X 0,Y 482.637,Z 375.28,A -85,B 0,C 180,E1 23258.881,E2 23258.881} C_VEL
LIN {X 0,Y 481.093,Z 372.23,A -85,B 0,C 180,E1 23258.343,E2 23258.343} C_VEL
LIN {X 0,Y 480.895,Z 371.148,A -85,B 0,C 180,E1 23258.169,E2 23258.169} C_VEL
LIN {X 0,Y 480.841,Z 371.127,A -85,B 0,C 180,E1 23254.733,E2 23254.733} C_VEL
LIN {X 0,Y 480.838,Z 371.147,A -85,B 0,C 180,E1 23251.062,E2 23251.062} C_VEL
LIN {X 0,Y 480.881,Z 371.131,A -85,B 0,C 180,E1 23247.624,E2 23247.624} C_VEL
LIN {X 0,Y 480.848,Z 371.116,A -85,B 0,C 180,E1 23244.115,E2 23244.115} C_VEL
LIN {X 0,Y 480.825,Z 371.15,A -85,B 0,C 180,E1 23240.667,E2 23240.667} C_VEL
LIN {X 0,Y 480.851,Z 371.115,A -85,B 0,C 180,E1 23237.173,E2 23237.173} C_VEL
LIN {X 0,Y 480.854,Z 371.152,A -85,B 0,C 180,E1 23233.712,E2 23233.712} C_VEL
LIN {X 0,Y 480.812,Z 371.153,A -85,B 0,C 180,E1 23230.302,E2 23230.302} C_VEL
LIN {X 0,Y 480.834,Z 371.15,A -85,B 0,C 180,E1 23226.807,E2 23226.807} C_VEL
LIN {X 0,Y 480.856,Z 371.152,A -85,B 0,C 180,E1 23223.337,E2 23223.337} C_VEL
LIN {X 0,Y 480.816,Z 371.153,A -85,B 0,C 180,E1 23219.881,E2 23219.881} C_VEL
LIN {X 0,Y 480.83,Z 371.151,A -85,B 0,C 180,E1 23216.304,E2 23216.304} C_VEL
LIN {X 0,Y 480.894,Z 371.147,A -85,B 0,C 180,E1 23212.833,E2 23212.833} C_VEL
LIN {X 0,Y 480.84,Z 371.152,A -85,B 0,C 180,E1 23209.335,E2 23209.335} C_VEL
LIN {X 0,Y 480.832,Z 371.151,A -85,B 0,C 180,E1 23205.796,E2 23205.796} C_VEL
LIN {X 0,Y 480.874,Z 371.111,A -85,B 0,C 180,E1 23202.328,E2 23202.328} C_VEL
LIN {X 0,Y 480.875,Z 371.148,A -85,B 0,C 180,E1 23198.79,E2 23198.79} C_VEL
LIN {X 0,Y 480.839,Z 371.124,A -85,B 0,C 180,E1 23195.294,E2 23195.294} C_VEL
LIN {X 0,Y 480.86,Z 371.134,A -85,B 0,C 180,E1 23191.7,E2 23191.7} C_VEL
LIN {X 0,Y 480.895,Z 371.143,A -85,B 0,C 180,E1 23188.241,E2 23188.241} C_VEL
LIN {X 0,Y 480.861,Z 371.12,A -85,B 0,C 180,E1 23184.686,E2 23184.686} C_VEL
LIN {X 0,Y 480.853,Z 371.124,A -85,B 0,C 180,E1 23181.1,E2 23181.1} C_VEL
LIN {X 0,Y 480.915,Z 371.285,A -85,B 0,C 180,E1 23179.897,E2 23179.897} C_VEL
LIN {X 0,Y 482.091,Z 374.452,A -85,B 0,C 180,E1 23179.658,E2 23179.658} C_VEL
LIN {X 0,Y 485.023,Z 377.679,A -85,B 0,C 180,E1 23179.175,E2 23179.175} C_VEL
LIN {X 0,Y 487.683,Z 381.558,A -85,B 0,C 180,E1 23178.726,E2 23178.726} C_VEL
LIN {X 0,Y 489.236,Z 383.425,A -85,B 0,C 180,E1 23178.476,E2 23178.476} C_VEL
LIN {X 0,Y 500.639,Z 399.145,A -85,B 0,C 180,E1 23176.684,E2 23176.684} C_VEL
LIN {X 0,Y 510.626,Z 413.547,A -85,B 0,C 180,E1 23175.212,E2 23175.212} C_VEL
LIN {X 0,Y 508.893,Z 491.597,A -85,B 0,C 180,E1 23173.886,E2 23173.886} C_VEL
LIN {X 0,Y 508.032,Z 499.297,A -85,B 0,C 180,E1 23173.832,E2 23173.832} C_VEL
LIN {X 0,Y 503.05,Z 519.919,A -85,B 0,C 180,E1 23173.981,E2 23173.981} C_VEL
LIN {X 0,Y 502.355,Z 526.529,A -85,B 0,C 180,E1 23173.929,E2 23173.929} C_VEL
LIN {X 0,Y 498.086,Z 710.89,A -85,B 0,C 180,E1 23170.811,E2 23170.811} C_VEL
LIN {X 0,Y 496.903,Z 733.823,A -85,B 0,C 180,E1 23170.238,E2 23170.238} C_VEL
LIN {X 0,Y 495.544,Z 753.789,A -85,B 0,C 180,E1 23169.566,E2 23169.566} C_VEL
LIN {X 0,Y 493.624,Z 776.244,A -85,B 0,C 180,E1 23168.593,E2 23168.593} C_VEL
LIN {X 0,Y 491.634,Z 796.39,A -85,B 0,C 180,E1 23167.518,E2 23167.518} C_VEL
LIN {X 0,Y 489.348,Z 816.936,A -85,B 0,C 180,E1 23166.187,E2 23166.187} C_VEL
LIN {X 0,Y 487.153,Z 835.366,A -85,B 0,C 180,E1 23164.786,E2 23164.786} C_VEL
LIN {X 0,Y 484.693,Z 854.866,A -85,B 0,C 180,E1 23163.063,E2 23163.063} C_VEL
LIN {X 0,Y 482.433,Z 873.104,A -85,B 0,C 180,E1 23161.203,E2 23161.203} C_VEL
LIN {X 0,Y 480.205,Z 890.312,A -85,B 0,C 180,E1 23159.154,E2 23159.154} C_VEL
LIN {X 0,Y 478.263,Z 906.338,A -85,B 0,C 180,E1 23156.975,E2 23156.975} C_VEL
LIN {X 0,Y 476.542,Z 920.952,A -85,B 0,C 180,E1 23154.676,E2 23154.676} C_VEL
LIN {X 0,Y 475.046,Z 934.973,A -85,B 0,C 180,E1 23152.13,E2 23152.13} C_VEL
LIN {X 0,Y 473.938,Z 946.973,A -85,B 0,C 180,E1 23149.597,E2 23149.597} C_VEL
LIN {X 0,Y 473.092,Z 957.536,A -85,B 0,C 180,E1 23146.955,E2 23146.955} C_VEL
LIN {X 0,Y 472.527,Z 966.605,A -85,B 0,C 180,E1 23144.276,E2 23144.276} C_VEL
LIN {X 0,Y 472.182,Z 973.849,A -85,B 0,C 180,E1 23141.603,E2 23141.603} C_VEL
LIN {X 0,Y 472.017,Z 979.735,A -85,B 0,C 180,E1 23138.894,E2 23138.894} C_VEL
LIN {X 0,Y 471.934,Z 983.901,A -85,B 0,C 180,E1 23136.202,E2 23136.202} C_VEL
LIN {X 0,Y 471.895,Z 986.688,A -85,B 0,C 180,E1 23133.522,E2 23133.522} C_VEL
LIN {X 0,Y 471.896,Z 987.818,A -85,B 0,C 180,E1 23130.971,E2 23130.971} C_VEL
LIN {X 0,Y 471.909,Z 987.722,A -85,B 0,C 180,E1 23128.422,E2 23128.422} C_VEL
LIN {X 0,Y 471.908,Z 985.998,A -85,B 0,C 180,E1 23125.626,E2 23125.626} C_VEL
LIN {X 0,Y 471.93,Z 983.22,A -85,B 0,C 180,E1 23123.187,E2 23123.187} C_VEL
LIN {X 0,Y 472.026,Z 978.431,A -85,B 0,C 180,E1 23120.368,E2 23120.368} C_VEL
LIN {X 0,Y 472.233,Z 972.856,A -85,B 0,C 180,E1 23117.901,E2 23117.901} C_VEL
LIN {X 0,Y 472.644,Z 964.705,A -85,B 0,C 180,E1 23115.045,E2 23115.045} C_VEL
LIN {X 0,Y 473.253,Z 955.554,A -85,B 0,C 180,E1 23112.417,E2 23112.417} C_VEL
LIN {X 0,Y 474.152,Z 944.501,A -85,B 0,C 180,E1 23109.77,E2 23109.77} C_VEL
LIN {X 0,Y 475.365,Z 932.2,A -85,B 0,C 180,E1 23107.233,E2 23107.233} C_VEL
LIN {X 0,Y 476.832,Z 918.39,A -85,B 0,C 180,E1 23104.81,E2 23104.81} C_VEL
LIN {X 0,Y 478.709,Z 902.437,A -85,B 0,C 180,E1 23102.378,E2 23102.378} C_VEL
LIN {X 0,Y 480.659,Z 886.918,A -85,B 0,C 180,E1 23100.328,E2 23100.328} C_VEL
LIN {X 0,Y 482.906,Z 869.028,A -85,B 0,C 180,E1 23098.274,E2 23098.274} C_VEL
LIN {X 0,Y 485.219,Z 851.042,A -85,B 0,C 180,E1 23096.483,E2 23096.483} C_VEL
LIN {X 0,Y 487.691,Z 830.753,A -85,B 0,C 180,E1 23094.755,E2 23094.755} C_VEL
LIN {X 0,Y 490.074,Z 810.777,A -85,B 0,C 180,E1 23093.293,E2 23093.293} C_VEL
LIN {X 0,Y 492.193,Z 790.996,A -85,B 0,C 180,E1 23092.088,E2 23092.088} C_VEL
LIN {X 0,Y 494.235,Z 769.944,A -85,B 0,C 180,E1 23091.016,E2 23091.016} C_VEL
LIN {X 0,Y 495.888,Z 748.755,A -85,B 0,C 180,E1 23090.158,E2 23090.158} C_VEL
LIN {X 0,Y 497.366,Z 725.605,A -85,B 0,C 180,E1 23089.438,E2 23089.438} C_VEL
LIN {X 0,Y 498.336,Z 703.723,A -85,B 0,C 180,E1 23088.965,E2 23088.965} C_VEL
LIN {X 0,Y 503.081,Z 495.042,A -85,B 0,C 180,E1 23085.445,E2 23085.445} C_VEL
LIN {X 0,Y 504.794,Z 416.991,A -85,B 0,C 180,E1 23084.09,E2 23084.09} C_VEL
LIN {X 0,Y 491.514,Z 398.087,A -85,B 0,C 180,E1 23082.05,E2 23082.05} C_VEL
LIN {X 0,Y 484.041,Z 388.03,A -85,B 0,C 180,E1 23080.827,E2 23080.827} C_VEL
LIN {X 0,Y 480.305,Z 383.022,A -85,B 0,C 180,E1 23080.19,E2 23080.19} C_VEL
LIN {X 0,Y 477.471,Z 379.221,A -85,B 0,C 180,E1 23079.694,E2 23079.694} C_VEL
LIN {X 0,Y 476.644,Z 377.904,A -85,B 0,C 180,E1 23079.543,E2 23079.543} C_VEL
LIN {X 0,Y 474.01,Z 375.253,A -85,B 0,C 180,E1 23079.09,E2 23079.09} C_VEL
LIN {X 0,Y 472.921,Z 372.107,A -85,B 0,C 180,E1 23078.849,E2 23078.849} C_VEL
LIN {X 0,Y 472.926,Z 372.107,A -85,B 0,C 180,E1 23075.252,E2 23075.252} C_VEL
LIN {X 0,Y 472.954,Z 372.134,A -85,B 0,C 180,E1 23071.583,E2 23071.583} C_VEL
LIN {X 0,Y 472.954,Z 372.118,A -85,B 0,C 180,E1 23067.922,E2 23067.922} C_VEL
LIN {X 0,Y 472.91,Z 372.109,A -85,B 0,C 180,E1 23064.335,E2 23064.335} C_VEL
LIN {X 0,Y 472.907,Z 372.141,A -85,B 0,C 180,E1 23060.676,E2 23060.676} C_VEL
LIN {X 0,Y 472.931,Z 372.097,A -85,B 0,C 180,E1 23057.09,E2 23057.09} C_VEL
LIN {X 0,Y 472.935,Z 372.137,A -85,B 0,C 180,E1 23053.572,E2 23053.572} C_VEL
LIN {X 0,Y 472.893,Z 372.14,A -85,B 0,C 180,E1 23050.107,E2 23050.107} C_VEL
LIN {X 0,Y 472.897,Z 372.14,A -85,B 0,C 180,E1 23046.434,E2 23046.434} C_VEL
LIN {X 0,Y 472.936,Z 372.14,A -85,B 0,C 180,E1 23042.909,E2 23042.909} C_VEL
LIN {X 0,Y 472.901,Z 372.139,A -85,B 0,C 180,E1 23039.395,E2 23039.395} C_VEL
LIN {X 0,Y 472.874,Z 372.142,A -85,B 0,C 180,E1 23035.878,E2 23035.878} C_VEL
LIN {X 0,Y 472.898,Z 372.142,A -85,B 0,C 180,E1 23032.346,E2 23032.346} C_VEL
LIN {X 0,Y 472.924,Z 372.14,A -85,B 0,C 180,E1 23028.779,E2 23028.779} C_VEL
LIN {X 0,Y 472.88,Z 372.143,A -85,B 0,C 180,E1 23025.302,E2 23025.302} C_VEL
LIN {X 0,Y 472.881,Z 372.111,A -85,B 0,C 180,E1 23021.637,E2 23021.637} C_VEL
LIN {X 0,Y 472.929,Z 372.129,A -85,B 0,C 180,E1 23018.129,E2 23018.129} C_VEL
LIN {X 0,Y 472.921,Z 372.127,A -85,B 0,C 180,E1 23014.584,E2 23014.584} C_VEL
LIN {X 0,Y 472.891,Z 372.111,A -85,B 0,C 180,E1 23011.074,E2 23011.074} C_VEL
LIN {X 0,Y 472.912,Z 372.131,A -85,B 0,C 180,E1 23007.511,E2 23007.511} C_VEL
LIN {X 0,Y 472.951,Z 372.135,A -85,B 0,C 180,E1 23004.005,E2 23004.005} C_VEL
LIN {X 0,Y 472.909,Z 372.176,A -85,B 0,C 180,E1 23002.887,E2 23002.887} C_VEL
LIN {X 0,Y 474.248,Z 375.615,A -85,B 0,C 180,E1 23002.309,E2 23002.309} C_VEL
LIN {X 0,Y 475.402,Z 377.274,A -85,B 0,C 180,E1 23001.959,E2 23001.959} C_VEL
LIN {X 0,Y 477.458,Z 381.288,A -85,B 0,C 180,E1 23001.234,E2 23001.234} C_VEL
LIN {X 0,Y 480.826,Z 388.079,A -85,B 0,C 180,E1 23000.104,E2 23000.104} C_VEL
LIN {X 0,Y 490.096,Z 401.431,A -85,B 0,C 180,E1 22998.546,E2 22998.546} C_VEL
LIN {X 0,Y 502.675,Z 420.69,A -85,B 0,C 180,E1 22996.57,E2 22996.57} C_VEL
LIN {X 0,Y 505.187,Z 425.041,A -85,B 0,C 180,E1 22996.185,E2 22996.185} C_VEL
LIN {X 0,Y 500.29,Z 638.335,A -85,B 0,C 180,E1 22992.568,E2 22992.568} C_VEL
LIN {X 0,Y 497.948,Z 740.001,A -85,B 0,C 180,E1 22990.85,E2 22990.85} C_VEL
LIN {X 0,Y 496.729,Z 762.811,A -85,B 0,C 180,E1 22990.28,E2 22990.28} C_VEL
LIN {X 0,Y 495.302,Z 783.851,A -85,B 0,C 180,E1 22989.572,E2 22989.572} C_VEL
LIN {X 0,Y 493.412,Z 805.924,A -85,B 0,C 180,E1 22988.614,E2 22988.614} C_VEL
LIN {X 0,Y 491.355,Z 827.41,A -85,B 0,C 180,E1 22987.472,E2 22987.472} C_VEL
LIN {X 0,Y 489.125,Z 847.998,A -85,B 0,C 180,E1 22986.135,E2 22986.135} C_VEL
LIN {X 0,Y 486.913,Z 867.468,A -85,B 0,C 180,E1 22984.663,E2 22984.663} C_VEL
LIN {X 0,Y 484.437,Z 886.932,A -85,B 0,C 180,E1 22982.91,E2 22982.91} C_VEL
LIN {X 0,Y 482.021,Z 906.132,A -85,B 0,C 180,E1 22980.902,E2 22980.902} C_VEL
LIN {X 0,Y 479.923,Z 922.667,A -85,B 0,C 180,E1 22978.901,E2 22978.901} C_VEL
LIN {X 0,Y 477.898,Z 939.155,A -85,B 0,C 180,E1 22976.595,E2 22976.595} C_VEL
LIN {X 0,Y 476.278,Z 953.52,A -85,B 0,C 180,E1 22974.294,E2 22974.294} C_VEL
LIN {X 0,Y 474.851,Z 966.912,A -85,B 0,C 180,E1 22971.786,E2 22971.786} C_VEL
LIN {X 0,Y 473.727,Z 979.3,A -85,B 0,C 180,E1 22969.094,E2 22969.094} C_VEL
LIN {X 0,Y 472.982,Z 989.07,A -85,B 0,C 180,E1 22966.58,E2 22966.58} C_VEL
LIN {X 0,Y 472.429,Z 998.299,A -85,B 0,C 180,E1 22963.729,E2 22963.729} C_VEL
LIN {X 0,Y 472.138,Z 1004.867,A -85,B 0,C 180,E1 22961.234,E2 22961.234} C_VEL
LIN {X 0,Y 471.995,Z 1010.642,A -85,B 0,C 180,E1 22958.401,E2 22958.401} C_VEL
LIN {X 0,Y 471.916,Z 1014.438,A -85,B 0,C 180,E1 22955.837,E2 22955.837} C_VEL
LIN {X 0,Y 471.887,Z 1016.986,A -85,B 0,C 180,E1 22953.036,E2 22953.036} C_VEL
LIN {X 0,Y 471.884,Z 1017.872,A -85,B 0,C 180,E1 22950.729,E2 22950.729} C_VEL
LIN {X 0,Y 471.909,Z 1017.594,A -85,B 0,C 180,E1 22948.058,E2 22948.058} C_VEL
LIN {X 0,Y 471.907,Z 1015.729,A -85,B 0,C 180,E1 22945.383,E2 22945.383} C_VEL
LIN {X 0,Y 471.934,Z 1012.496,A -85,B 0,C 180,E1 22942.698,E2 22942.698} C_VEL
LIN {X 0,Y 472.035,Z 1007.831,A -85,B 0,C 180,E1 22940.122,E2 22940.122} C_VEL
LIN {X 0,Y 472.28,Z 1001.831,A -85,B 0,C 180,E1 22937.531,E2 22937.531} C_VEL
LIN {X 0,Y 472.701,Z 993.752,A -85,B 0,C 180,E1 22934.796,E2 22934.796} C_VEL
LIN {X 0,Y 473.341,Z 984.454,A -85,B 0,C 180,E1 22932.167,E2 22932.167} C_VEL
LIN {X 0,Y 474.267,Z 973.161,A -85,B 0,C 180,E1 22929.518,E2 22929.518} C_VEL
LIN {X 0,Y 475.582,Z 959.866,A -85,B 0,C 180,E1 22926.853,E2 22926.853} C_VEL
LIN {X 0,Y 477.055,Z 946.592,A -85,B 0,C 180,E1 22924.558,E2 22924.558} C_VEL
LIN {X 0,Y 478.907,Z 930.745,A -85,B 0,C 180,E1 22922.189,E2 22922.189} C_VEL
LIN {X 0,Y 481.05,Z 913.928,A -85,B 0,C 180,E1 22920,E2 22920} C_VEL
LIN {X 0,Y 483.265,Z 896.206,A -85,B 0,C 180,E1 22918.022,E2 22918.022} C_VEL
LIN {X 0,Y 485.788,Z 876.294,A -85,B 0,C 180,E1 22916.103,E2 22916.103} C_VEL
LIN {X 0,Y 487.889,Z 858.737,A -85,B 0,C 180,E1 22914.65,E2 22914.65} C_VEL
LIN {X 0,Y 490.269,Z 837.62,A -85,B 0,C 180,E1 22913.165,E2 22913.165} C_VEL
LIN {X 0,Y 492.264,Z 818.313,A -85,B 0,C 180,E1 22912.022,E2 22912.022} C_VEL
LIN {X 0,Y 494.304,Z 795.726,A -85,B 0,C 180,E1 22910.915,E2 22910.915} C_VEL
LIN {X 0,Y 495.957,Z 774.438,A -85,B 0,C 180,E1 22910.085,E2 22910.085} C_VEL
LIN {X 0,Y 497.394,Z 751.302,A -85,B 0,C 180,E1 22909.409,E2 22909.409} C_VEL
LIN {X 0,Y 498.342,Z 728.818,A -85,B 0,C 180,E1 22908.941,E2 22908.941} C_VEL
LIN {X 0,Y 502.913,Z 520.832,A -85,B 0,C 180,E1 22905.449,E2 22905.449} C_VEL
LIN {X 0,Y 505.104,Z 424.544,A -85,B 0,C 180,E1 22903.795,E2 22903.795} C_VEL
LIN {X 0,Y 491.704,Z 403.813,A -85,B 0,C 180,E1 22901.716,E2 22901.716} C_VEL
LIN {X 0,Y 481.983,Z 389.705,A -85,B 0,C 180,E1 22900.099,E2 22900.099} C_VEL
LIN {X 0,Y 480.2,Z 386.868,A -85,B 0,C 180,E1 22899.734,E2 22899.734} C_VEL
LIN {X 0,Y 476.649,Z 380.167,A -85,B 0,C 180,E1 22898.536,E2 22898.536} C_VEL
LIN {X 0,Y 474.759,Z 376.29,A -85,B 0,C 180,E1 22897.846,E2 22897.846} C_VEL
LIN {X 0,Y 473.238,Z 373.614,A -85,B 0,C 180,E1 22897.327,E2 22897.327} C_VEL
LIN {X 0,Y 472.905,Z 372.138,A -85,B 0,C 180,E1 22897.112,E2 22897.112} C_VEL
LIN {X 0,Y 472.927,Z 372.109,A -85,B 0,C 180,E1 22893.603,E2 22893.603} C_VEL
LIN {X 0,Y 472.939,Z 372.107,A -85,B 0,C 180,E1 22890.069,E2 22890.069} C_VEL
LIN {X 0,Y 472.895,Z 372.138,A -85,B 0,C 180,E1 22886.587,E2 22886.587} C_VEL
LIN {X 0,Y 472.889,Z 372.109,A -85,B 0,C 180,E1 22882.895,E2 22882.895} C_VEL
LIN {X 0,Y 472.938,Z 372.122,A -85,B 0,C 180,E1 22879.474,E2 22879.474} C_VEL
LIN {X 0,Y 472.905,Z 372.122,A -85,B 0,C 180,E1 22875.87,E2 22875.87} C_VEL
LIN {X 0,Y 472.875,Z 372.133,A -85,B 0,C 180,E1 22872.381,E2 22872.381} C_VEL
LIN {X 0,Y 472.897,Z 372.134,A -85,B 0,C 180,E1 22868.879,E2 22868.879} C_VEL
LIN {X 0,Y 472.908,Z 372.132,A -85,B 0,C 180,E1 22865.459,E2 22865.459} C_VEL
LIN {X 0,Y 472.874,Z 372.133,A -85,B 0,C 180,E1 22861.938,E2 22861.938} C_VEL
LIN {X 0,Y 472.884,Z 372.133,A -85,B 0,C 180,E1 22858.303,E2 22858.303} C_VEL
LIN {X 0,Y 472.936,Z 372.129,A -85,B 0,C 180,E1 22854.784,E2 22854.784} C_VEL
LIN {X 0,Y 472.899,Z 372.134,A -85,B 0,C 180,E1 22851.366,E2 22851.366} C_VEL
LIN {X 0,Y 472.891,Z 372.132,A -85,B 0,C 180,E1 22847.793,E2 22847.793} C_VEL
LIN {X 0,Y 472.927,Z 372.122,A -85,B 0,C 180,E1 22844.299,E2 22844.299} C_VEL
LIN {X 0,Y 472.938,Z 372.119,A -85,B 0,C 180,E1 22840.743,E2 22840.743} C_VEL
LIN {X 0,Y 472.902,Z 372.114,A -85,B 0,C 180,E1 22837.237,E2 22837.237} C_VEL
LIN {X 0,Y 472.908,Z 372.139,A -85,B 0,C 180,E1 22833.505,E2 22833.505} C_VEL
LIN {X 0,Y 472.958,Z 372.101,A -85,B 0,C 180,E1 22830.071,E2 22830.071} C_VEL
LIN {X 0,Y 472.945,Z 372.114,A -85,B 0,C 180,E1 22826.393,E2 22826.393} C_VEL
LIN {X 0,Y 472.922,Z 372.141,A -85,B 0,C 180,E1 22822.795,E2 22822.795} C_VEL
LIN {X 0,Y 472.929,Z 372.219,A -85,B 0,C 180,E1 22821.05,E2 22821.05} C_VEL
LIN {X 0,Y 474.06,Z 375.344,A -85,B 0,C 180,E1 22820.806,E2 22820.806} C_VEL
LIN {X 0,Y 476.581,Z 377.867,A -85,B 0,C 180,E1 22820.373,E2 22820.373} C_VEL
LIN {X 0,Y 477.752,Z 379.752,A -85,B 0,C 180,E1 22820.158,E2 22820.158} C_VEL
LIN {X 0,Y 480.692,Z 383.379,A -85,B 0,C 180,E1 22819.653,E2 22819.653} C_VEL
LIN {X 0,Y 484.58,Z 388.587,A -85,B 0,C 180,E1 22818.993,E2 22818.993} C_VEL
LIN {X 0,Y 496.608,Z 405.254,A -85,B 0,C 180,E1 22817.056,E2 22817.056} C_VEL
LIN {X 0,Y 504.937,Z 417.397,A -85,B 0,C 180,E1 22815.795,E2 22815.795} C_VEL
LIN {X 0,Y 502.355,Z 526.529,A -85,B 0,C 180,E1 22813.929,E2 22813.929} C_VEL
LIN {X 0,Y 501.456,Z 534.231,A -85,B 0,C 180,E1 22813.878,E2 22813.878} C_VEL
LIN {X 0,Y 496.448,Z 554.843,A -85,B 0,C 180,E1 22814.032,E2 22814.032} C_VEL
LIN {X 0,Y 495.762,Z 561.449,A -85,B 0,C 180,E1 22813.979,E2 22813.979} C_VEL
LIN {X 0,Y 492.051,Z 711.463,A -85,B 0,C 180,E1 22811.415,E2 22811.415} C_VEL
LIN {X 0,Y 490.8,Z 734.292,A -85,B 0,C 180,E1 22810.839,E2 22810.839} C_VEL
LIN {X 0,Y 489.326,Z 754.77,A -85,B 0,C 180,E1 22810.141,E2 22810.141} C_VEL
LIN {X 0,Y 487.348,Z 776.562,A -85,B 0,C 180,E1 22809.185,E2 22809.185} C_VEL
LIN {X 0,Y 485.271,Z 796.366,A -85,B 0,C 180,E1 22808.12,E2 22808.12} C_VEL
LIN {X 0,Y 482.795,Z 817.252,A -85,B 0,C 180,E1 22806.758,E2 22806.758} C_VEL
LIN {X 0,Y 480.374,Z 836.404,A -85,B 0,C 180,E1 22805.284,E2 22805.284} C_VEL
LIN {X 0,Y 477.704,Z 855.626,A -85,B 0,C 180,E1 22803.538,E2 22803.538} C_VEL
LIN {X 0,Y 475.019,Z 875.35,A -85,B 0,C 180,E1 22801.463,E2 22801.463} C_VEL
LIN {X 0,Y 472.748,Z 891.838,A -85,B 0,C 180,E1 22799.451,E2 22799.451} C_VEL
LIN {X 0,Y 470.498,Z 908.879,A -85,B 0,C 180,E1 22797.047,E2 22797.047} C_VEL
LIN {X 0,Y 468.69,Z 923.561,A -85,B 0,C 180,E1 22794.661,E2 22794.661} C_VEL
LIN {X 0,Y 467.143,Z 936.88,A -85,B 0,C 180,E1 22792.127,E2 22792.127} C_VEL
LIN {X 0,Y 465.931,Z 949.128,A -85,B 0,C 180,E1 22789.425,E2 22789.425} C_VEL
LIN {X 0,Y 465.11,Z 958.913,A -85,B 0,C 180,E1 22786.868,E2 22786.868} C_VEL
LIN {X 0,Y 464.509,Z 967.873,A -85,B 0,C 180,E1 22784.075,E2 22784.075} C_VEL
LIN {X 0,Y 464.187,Z 974.456,A -85,B 0,C 180,E1 22781.554,E2 22781.554} C_VEL
LIN {X 0,Y 464.009,Z 980.357,A -85,B 0,C 180,E1 22778.674,E2 22778.674} C_VEL
LIN {X 0,Y 463.927,Z 984.221,A -85,B 0,C 180,E1 22776.061,E2 22776.061} C_VEL
LIN {X 0,Y 463.886,Z 986.892,A -85,B 0,C 180,E1 22773.212,E2 22773.212} C_VEL
LIN {X 0,Y 463.887,Z 987.864,A -85,B 0,C 180,E1 22770.741,E2 22770.741} C_VEL
LIN {X 0,Y 463.911,Z 987.619,A -85,B 0,C 180,E1 22768.024,E2 22768.024} C_VEL
LIN {X 0,Y 463.905,Z 985.77,A -85,B 0,C 180,E1 22765.302,E2 22765.302} C_VEL
LIN {X 0,Y 463.937,Z 982.568,A -85,B 0,C 180,E1 22762.571,E2 22762.571} C_VEL
LIN {X 0,Y 464.049,Z 977.921,A -85,B 0,C 180,E1 22759.95,E2 22759.95} C_VEL
LIN {X 0,Y 464.322,Z 971.873,A -85,B 0,C 180,E1 22757.285,E2 22757.285} C_VEL
LIN {X 0,Y 464.774,Z 963.891,A -85,B 0,C 180,E1 22754.53,E2 22754.53} C_VEL
LIN {X 0,Y 465.471,Z 954.619,A -85,B 0,C 180,E1 22751.854,E2 22751.854} C_VEL
LIN {X 0,Y 466.485,Z 943.311,A -85,B 0,C 180,E1 22749.151,E2 22749.151} C_VEL
LIN {X 0,Y 467.908,Z 930.096,A -85,B 0,C 180,E1 22746.45,E2 22746.45} C_VEL
LIN {X 0,Y 469.509,Z 916.842,A -85,B 0,C 180,E1 22744.118,E2 22744.118} C_VEL
LIN {X 0,Y 471.513,Z 901.04,A -85,B 0,C 180,E1 22741.713,E2 22741.713} C_VEL
LIN {X 0,Y 473.797,Z 884.367,A -85,B 0,C 180,E1 22739.504,E2 22739.504} C_VEL
LIN {X 0,Y 476.198,Z 866.585,A -85,B 0,C 180,E1 22737.489,E2 22737.489} C_VEL
LIN {X 0,Y 479.015,Z 846.215,A -85,B 0,C 180,E1 22735.483,E2 22735.483} C_VEL
LIN {X 0,Y 481.466,Z 827.838,A -85,B 0,C 180,E1 22733.937,E2 22733.937} C_VEL
LIN {X 0,Y 484.043,Z 807.085,A -85,B 0,C 180,E1 22732.461,E2 22732.461} C_VEL
LIN {X 0,Y 486.212,Z 787.921,A -85,B 0,C 180,E1 22731.311,E2 22731.311} C_VEL
LIN {X 0,Y 488.335,Z 765.817,A -85,B 0,C 180,E1 22730.225,E2 22730.225} C_VEL
LIN {X 0,Y 490.189,Z 743.652,A -85,B 0,C 180,E1 22729.361,E2 22729.361} C_VEL
LIN {X 0,Y 491.537,Z 721.828,A -85,B 0,C 180,E1 22728.733,E2 22728.733} C_VEL
LIN {X 0,Y 492.519,Z 698.447,A -85,B 0,C 180,E1 22728.251,E2 22728.251} C_VEL
LIN {X 0,Y 497.576,Z 488.659,A -85,B 0,C 180,E1 22724.684,E2 22724.684} C_VEL
LIN {X 0,Y 499.197,Z 420.945,A -85,B 0,C 180,E1 22723.498,E2 22723.498} C_VEL
LIN {X 0,Y 487.328,Z 403.926,A -85,B 0,C 180,E1 22721.624,E2 22721.624} C_VEL
LIN {X 0,Y 479.784,Z 393.761,A -85,B 0,C 180,E1 22720.361,E2 22720.361} C_VEL
LIN {X 0,Y 476.228,Z 389.016,A -85,B 0,C 180,E1 22719.74,E2 22719.74} C_VEL
LIN {X 0,Y 472.728,Z 384.29,A -85,B 0,C 180,E1 22719.111,E2 22719.111} C_VEL
LIN {X 0,Y 469.803,Z 380.628,A -85,B 0,C 180,E1 22718.578,E2 22718.578} C_VEL
LIN {X 0,Y 468.73,Z 378.91,A -85,B 0,C 180,E1 22718.37,E2 22718.37} C_VEL
LIN {X 0,Y 466.141,Z 376.313,A -85,B 0,C 180,E1 22717.899,E2 22717.899} C_VEL
LIN {X 0,Y 465.017,Z 373.176,A -85,B 0,C 180,E1 22717.641,E2 22717.641} C_VEL
LIN {X 0,Y 465.015,Z 373.09,A -85,B 0,C 180,E1 22713.914,E2 22713.914} C_VEL
LIN {X 0,Y 464.985,Z 373.1,A -85,B 0,C 180,E1 22710.353,E2 22710.353} C_VEL
LIN {X 0,Y 464.974,Z 373.129,A -85,B 0,C 180,E1 22706.707,E2 22706.707} C_VEL
LIN {X 0,Y 464.981,Z 373.09,A -85,B 0,C 180,E1 22703.039,E2 22703.039} C_VEL
LIN {X 0,Y 465.014,Z 373.117,A -85,B 0,C 180,E1 22699.468,E2 22699.468} C_VEL
LIN {X 0,Y 464.976,Z 373.098,A -85,B 0,C 180,E1 22695.849,E2 22695.849} C_VEL
LIN {X 0,Y 464.956,Z 373.121,A -85,B 0,C 180,E1 22692.292,E2 22692.292} C_VEL
LIN {X 0,Y 464.978,Z 373.119,A -85,B 0,C 180,E1 22688.782,E2 22688.782} C_VEL
LIN {X 0,Y 464.991,Z 373.12,A -85,B 0,C 180,E1 22685.306,E2 22685.306} C_VEL
LIN {X 0,Y 464.948,Z 373.127,A -85,B 0,C 180,E1 22681.726,E2 22681.726} C_VEL
LIN {X 0,Y 464.939,Z 373.124,A -85,B 0,C 180,E1 22678.028,E2 22678.028} C_VEL
LIN {X 0,Y 464.965,Z 373.119,A -85,B 0,C 180,E1 22674.447,E2 22674.447} C_VEL
LIN {X 0,Y 464.968,Z 373.123,A -85,B 0,C 180,E1 22670.969,E2 22670.969} C_VEL
LIN {X 0,Y 464.936,Z 373.126,A -85,B 0,C 180,E1 22667.456,E2 22667.456} C_VEL
LIN {X 0,Y 464.943,Z 373.115,A -85,B 0,C 180,E1 22663.766,E2 22663.766} C_VEL
LIN {X 0,Y 464.994,Z 373.116,A -85,B 0,C 180,E1 22660.27,E2 22660.27} C_VEL
LIN {X 0,Y 464.965,Z 373.098,A -85,B 0,C 180,E1 22656.827,E2 22656.827} C_VEL
LIN {X 0,Y 464.954,Z 373.132,A -85,B 0,C 180,E1 22653.292,E2 22653.292} C_VEL
LIN {X 0,Y 464.985,Z 373.102,A -85,B 0,C 180,E1 22649.79,E2 22649.79} C_VEL
LIN {X 0,Y 464.995,Z 373.094,A -85,B 0,C 180,E1 22646.306,E2 22646.306} C_VEL
LIN {X 0,Y 465.022,Z 373.198,A -85,B 0,C 180,E1 22644.019,E2 22644.019} C_VEL
LIN {X 0,Y 466.333,Z 376.681,A -85,B 0,C 180,E1 22643.413,E2 22643.413} C_VEL
LIN {X 0,Y 467.478,Z 378.235,A -85,B 0,C 180,E1 22643.058,E2 22643.058} C_VEL
LIN {X 0,Y 469.464,Z 382.142,A -85,B 0,C 180,E1 22642.321,E2 22642.321} C_VEL
LIN {X 0,Y 472.387,Z 387.667,A -85,B 0,C 180,E1 22641.343,E2 22641.343} C_VEL
LIN {X 0,Y 485.492,Z 406.489,A -85,B 0,C 180,E1 22639.048,E2 22639.048} C_VEL
LIN {X 0,Y 498.672,Z 426.962,A -85,B 0,C 180,E1 22636.925,E2 22636.925} C_VEL
LIN {X 0,Y 499.533,Z 428.837,A -85,B 0,C 180,E1 22636.782,E2 22636.782} C_VEL
LIN {X 0,Y 494.32,Z 641.096,A -85,B 0,C 180,E1 22633.148,E2 22633.148} C_VEL
LIN {X 0,Y 491.881,Z 739.806,A -85,B 0,C 180,E1 22631.462,E2 22631.462} C_VEL
LIN {X 0,Y 490.577,Z 762.627,A -85,B 0,C 180,E1 22630.887,E2 22630.887} C_VEL
LIN {X 0,Y 489.005,Z 784.403,A -85,B 0,C 180,E1 22630.147,E2 22630.147} C_VEL
LIN {X 0,Y 487.062,Z 805.618,A -85,B 0,C 180,E1 22629.213,E2 22629.213} C_VEL
LIN {X 0,Y 484.97,Z 825.963,A -85,B 0,C 180,E1 22628.127,E2 22628.127} C_VEL
LIN {X 0,Y 482.567,Z 846.779,A -85,B 0,C 180,E1 22626.779,E2 22626.779} C_VEL
LIN {X 0,Y 480.108,Z 867.185,A -85,B 0,C 180,E1 22625.227,E2 22625.227} C_VEL
LIN {X 0,Y 477.532,Z 886.57,A -85,B 0,C 180,E1 22623.481,E2 22623.481} C_VEL
LIN {X 0,Y 475.213,Z 904.034,A -85,B 0,C 180,E1 22621.661,E2 22621.661} C_VEL
LIN {X 0,Y 472.841,Z 921.146,A -85,B 0,C 180,E1 22619.584,E2 22619.584} C_VEL
LIN {X 0,Y 470.576,Z 938.308,A -85,B 0,C 180,E1 22617.179,E2 22617.179} C_VEL
LIN {X 0,Y 468.779,Z 952.749,A -85,B 0,C 180,E1 22614.843,E2 22614.843} C_VEL
LIN {X 0,Y 467.262,Z 965.82,A -85,B 0,C 180,E1 22612.386,E2 22612.386} C_VEL
LIN {X 0,Y 466.08,Z 977.732,A -85,B 0,C 180,E1 22609.811,E2 22609.811} C_VEL
LIN {X 0,Y 465.17,Z 988.151,A -85,B 0,C 180,E1 22607.124,E2 22607.124} C_VEL
LIN {X 0,Y 464.55,Z 997.286,A -85,B 0,C 180,E1 22604.329,E2 22604.329} C_VEL
LIN {X 0,Y 464.213,Z 1003.958,A -85,B 0,C 180,E1 22601.806,E2 22601.806} C_VEL
LIN {X 0,Y 464.024,Z 1009.81,A -85,B 0,C 180,E1 22599.049,E2 22599.049} C_VEL
LIN {X 0,Y 463.941,Z 1013.96,A -85,B 0,C 180,E1 22596.31,E2 22596.31} C_VEL
LIN {X 0,Y 463.896,Z 1016.713,A -85,B 0,C 180,E1 22593.584,E2 22593.584} C_VEL
LIN {X 0,Y 463.892,Z 1017.826,A -85,B 0,C 180,E1 22590.988,E2 22590.988} C_VEL
LIN {X 0,Y 463.907,Z 1017.713,A -85,B 0,C 180,E1 22588.395,E2 22588.395} C_VEL
LIN {X 0,Y 463.908,Z 1015.956,A -85,B 0,C 180,E1 22585.551,E2 22585.551} C_VEL
LIN {X 0,Y 463.928,Z 1013.162,A -85,B 0,C 180,E1 22583.069,E2 22583.069} C_VEL
LIN {X 0,Y 464.038,Z 1008.339,A -85,B 0,C 180,E1 22580.201,E2 22580.201} C_VEL
LIN {X 0,Y 464.274,Z 1002.746,A -85,B 0,C 180,E1 22577.692,E2 22577.692} C_VEL
LIN {X 0,Y 464.733,Z 994.56,A -85,B 0,C 180,E1 22574.785,E2 22574.785} C_VEL
LIN {X 0,Y 465.406,Z 985.397,A -85,B 0,C 180,E1 22572.111,E2 22572.111} C_VEL
LIN {X 0,Y 466.389,Z 974.306,A -85,B 0,C 180,E1 22569.418,E2 22569.418} C_VEL
LIN {X 0,Y 467.739,Z 961.779,A -85,B 0,C 180,E1 22566.806,E2 22566.806} C_VEL
LIN {X 0,Y 469.338,Z 948.131,A -85,B 0,C 180,E1 22564.38,E2 22564.38} C_VEL
LIN {X 0,Y 471.429,Z 931.669,A -85,B 0,C 180,E1 22561.846,E2 22561.846} C_VEL
LIN {X 0,Y 473.624,Z 915.578,A -85,B 0,C 180,E1 22559.703,E2 22559.703} C_VEL
LIN {X 0,Y 475.992,Z 898.029,A -85,B 0,C 180,E1 22557.688,E2 22557.688} C_VEL
LIN {X 0,Y 478.283,Z 881.164,A -85,B 0,C 180,E1 22556.003,E2 22556.003} C_VEL
LIN {X 0,Y 480.77,Z 861.461,A -85,B 0,C 180,E1 22554.318,E2 22554.318} C_VEL
LIN {X 0,Y 483.253,Z 841.335,A -85,B 0,C 180,E1 22552.838,E2 22552.838} C_VEL
LIN {X 0,Y 485.455,Z 821.423,A -85,B 0,C 180,E1 22551.618,E2 22551.618} C_VEL
LIN {X 0,Y 487.597,Z 800.461,A -85,B 0,C 180,E1 22550.535,E2 22550.535} C_VEL
LIN {X 0,Y 489.459,Z 777.949,A -85,B 0,C 180,E1 22549.614,E2 22549.614} C_VEL
LIN {X 0,Y 491.084,Z 754.91,A -85,B 0,C 180,E1 22548.891,E2 22548.891} C_VEL
LIN {X 0,Y 492.148,Z 732.651,A -85,B 0,C 180,E1 22548.404,E2 22548.404} C_VEL
LIN {X 0,Y 497.081,Z 525.535,A -85,B 0,C 180,E1 22544.884,E2 22544.884} C_VEL
LIN {X 0,Y 499.419,Z 428.185,A -85,B 0,C 180,E1 22543.192,E2 22543.192} C_VEL
LIN {X 0,Y 487.141,Z 409.087,A -85,B 0,C 180,E1 22541.232,E2 22541.232} C_VEL
LIN {X 0,Y 477.966,Z 395.631,A -85,B 0,C 180,E1 22539.666,E2 22539.666} C_VEL
LIN {X 0,Y 471.83,Z 386.757,A -85,B 0,C 180,E1 22538.536,E2 22538.536} C_VEL
LIN {X 0,Y 468.914,Z 381.416,A -85,B 0,C 180,E1 22537.523,E2 22537.523} C_VEL
LIN {X 0,Y 467.1,Z 377.64,A -85,B 0,C 180,E1 22536.823,E2 22536.823} C_VEL
LIN {X 0,Y 465.366,Z 374.704,A -85,B 0,C 180,E1 22536.217,E2 22536.217} C_VEL
LIN {X 0,Y 465.012,Z 373.12,A -85,B 0,C 180,E1 22535.944,E2 22535.944} C_VEL
LIN {X 0,Y 464.986,Z 373.122,A -85,B 0,C 180,E1 22532.332,E2 22532.332} C_VEL
LIN {X 0,Y 464.953,Z 373.094,A -85,B 0,C 180,E1 22528.796,E2 22528.796} C_VEL
LIN {X 0,Y 464.968,Z 373.108,A -85,B 0,C 180,E1 22525.199,E2 22525.199} C_VEL
LIN {X 0,Y 465.01,Z 373.11,A -85,B 0,C 180,E1 22521.705,E2 22521.705} C_VEL
LIN {X 0,Y 464.953,Z 373.092,A -85,B 0,C 180,E1 22518.124,E2 22518.124} C_VEL
LIN {X 0,Y 464.942,Z 373.132,A -85,B 0,C 180,E1 22514.572,E2 22514.572} C_VEL
LIN {X 0,Y 464.971,Z 373.131,A -85,B 0,C 180,E1 22511.033,E2 22511.033} C_VEL
LIN {X 0,Y 464.981,Z 373.129,A -85,B 0,C 180,E1 22507.413,E2 22507.413} C_VEL
LIN {X 0,Y 464.94,Z 373.132,A -85,B 0,C 180,E1 22503.822,E2 22503.822} C_VEL
LIN {X 0,Y 464.94,Z 373.131,A -85,B 0,C 180,E1 22500.246,E2 22500.246} C_VEL
LIN {X 0,Y 464.99,Z 373.13,A -85,B 0,C 180,E1 22496.795,E2 22496.795} C_VEL
LIN {X 0,Y 464.976,Z 373.128,A -85,B 0,C 180,E1 22493.208,E2 22493.208} C_VEL
LIN {X 0,Y 464.949,Z 373.129,A -85,B 0,C 180,E1 22489.718,E2 22489.718} C_VEL
LIN {X 0,Y 464.965,Z 373.129,A -85,B 0,C 180,E1 22486.063,E2 22486.063} C_VEL
LIN {X 0,Y 465.005,Z 373.083,A -85,B 0,C 180,E1 22482.609,E2 22482.609} C_VEL
LIN {X 0,Y 464.974,Z 373.13,A -85,B 0,C 180,E1 22479.086,E2 22479.086} C_VEL
LIN {X 0,Y 464.961,Z 373.095,A -85,B 0,C 180,E1 22475.438,E2 22475.438} C_VEL
LIN {X 0,Y 464.99,Z 373.109,A -85,B 0,C 180,E1 22471.825,E2 22471.825} C_VEL
LIN {X 0,Y 465.018,Z 373.12,A -85,B 0,C 180,E1 22468.211,E2 22468.211} C_VEL
LIN {X 0,Y 464.995,Z 373.095,A -85,B 0,C 180,E1 22464.509,E2 22464.509} C_VEL
LIN {X 0,Y 465.04,Z 373.325,A -85,B 0,C 180,E1 22462.254,E2 22462.254} C_VEL
LIN {X 0,Y 466.208,Z 376.419,A -85,B 0,C 180,E1 22461.991,E2 22461.991} C_VEL
LIN {X 0,Y 468.661,Z 378.876,A -85,B 0,C 180,E1 22461.545,E2 22461.545} C_VEL
LIN {X 0,Y 469.741,Z 380.528,A -85,B 0,C 180,E1 22461.338,E2 22461.338} C_VEL
LIN {X 0,Y 472.519,Z 384.111,A -85,B 0,C 180,E1 22460.829,E2 22460.829} C_VEL
LIN {X 0,Y 473.857,Z 385.763,A -85,B 0,C 180,E1 22460.59,E2 22460.59} C_VEL
LIN {X 0,Y 485.306,Z 401.1,A -85,B 0,C 180,E1 22458.617,E2 22458.617} C_VEL
LIN {X 0,Y 498.154,Z 419.338,A -85,B 0,C 180,E1 22456.572,E2 22456.572} C_VEL
LIN {X 0,Y 499.292,Z 421.525,A -85,B 0,C 180,E1 22456.388,E2 22456.388} C_VEL
LIN {X 0,Y 495.762,Z 561.449,A -85,B 0,C 180,E1 22453.979,E2 22453.979} C_VEL
LIN {X 0,Y 494.875,Z 569.149,A -85,B 0,C 180,E1 22453.926,E2 22453.926} C_VEL
LIN {X 0,Y 489.855,Z 589.759,A -85,B 0,C 180,E1 22454.085,E2 22454.085} C_VEL
LIN {X 0,Y 489.144,Z 596.368,A -85,B 0,C 180,E1 22454.033,E2 22454.033} C_VEL
LIN {X 0,Y 486.072,Z 712.028,A -85,B 0,C 180,E1 22452.035,E2 22452.035} C_VEL
LIN {X 0,Y 484.753,Z 734.761,A -85,B 0,C 180,E1 22451.454,E2 22451.454} C_VEL
LIN {X 0,Y 483.169,Z 755.644,A -85,B 0,C 180,E1 22450.734,E2 22450.734} C_VEL
LIN {X 0,Y 481.045,Z 777.6,A -85,B 0,C 180,E1 22449.756,E2 22449.756} C_VEL
LIN {X 0,Y 478.77,Z 798.123,A -85,B 0,C 180,E1 22448.635,E2 22448.635} C_VEL
LIN {X 0,Y 476.153,Z 818.667,A -85,B 0,C 180,E1 22447.264,E2 22447.264} C_VEL
LIN {X 0,Y 473.505,Z 838.37,A -85,B 0,C 180,E1 22445.717,E2 22445.717} C_VEL
LIN {X 0,Y 470.69,Z 857.261,A -85,B 0,C 180,E1 22443.959,E2 22443.959} C_VEL
LIN {X 0,Y 467.953,Z 875.615,A -85,B 0,C 180,E1 22441.977,E2 22441.977} C_VEL
LIN {X 0,Y 465.167,Z 894.376,A -85,B 0,C 180,E1 22439.624,E2 22439.624} C_VEL
LIN {X 0,Y 462.97,Z 909.728,A -85,B 0,C 180,E1 22437.384,E2 22437.384} C_VEL
LIN {X 0,Y 461.04,Z 924.239,A -85,B 0,C 180,E1 22434.971,E2 22434.971} C_VEL
LIN {X 0,Y 459.459,Z 936.882,A -85,B 0,C 180,E1 22432.517,E2 22432.517} C_VEL
LIN {X 0,Y 458.139,Z 949.132,A -85,B 0,C 180,E1 22429.769,E2 22429.769} C_VEL
LIN {X 0,Y 457.227,Z 959.04,A -85,B 0,C 180,E1 22427.132,E2 22427.132} C_VEL
LIN {X 0,Y 456.551,Z 968.228,A -85,B 0,C 180,E1 22424.197,E2 22424.197} C_VEL
LIN {X 0,Y 456.207,Z 974.761,A -85,B 0,C 180,E1 22421.631,E2 22421.631} C_VEL
LIN {X 0,Y 456.013,Z 980.565,A -85,B 0,C 180,E1 22418.7,E2 22418.7} C_VEL
LIN {X 0,Y 455.933,Z 984.222,A -85,B 0,C 180,E1 22416.168,E2 22416.168} C_VEL
LIN {X 0,Y 455.886,Z 986.893,A -85,B 0,C 180,E1 22413.268,E2 22413.268} C_VEL
LIN {X 0,Y 455.888,Z 987.864,A -85,B 0,C 180,E1 22410.754,E2 22410.754} C_VEL
LIN {X 0,Y 455.911,Z 987.619,A -85,B 0,C 180,E1 22407.989,E2 22407.989} C_VEL
LIN {X 0,Y 455.905,Z 985.883,A -85,B 0,C 180,E1 22405.346,E2 22405.346} C_VEL
LIN {X 0,Y 455.933,Z 982.898,A -85,B 0,C 180,E1 22402.693,E2 22402.693} C_VEL
LIN {X 0,Y 456.062,Z 978.092,A -85,B 0,C 180,E1 22399.859,E2 22399.859} C_VEL
LIN {X 0,Y 456.354,Z 972.103,A -85,B 0,C 180,E1 22397.157,E2 22397.157} C_VEL
LIN {X 0,Y 456.838,Z 964.238,A -85,B 0,C 180,E1 22394.367,E2 22394.367} C_VEL
LIN {X 0,Y 457.629,Z 954.616,A -85,B 0,C 180,E1 22391.532,E2 22391.532} C_VEL
LIN {X 0,Y 458.678,Z 943.846,A -85,B 0,C 180,E1 22388.905,E2 22388.905} C_VEL
LIN {X 0,Y 460.124,Z 931.49,A -85,B 0,C 180,E1 22386.299,E2 22386.299} C_VEL
LIN {X 0,Y 461.803,Z 918.376,A -85,B 0,C 180,E1 22383.93,E2 22383.93} C_VEL
LIN {X 0,Y 463.995,Z 902.422,A -85,B 0,C 180,E1 22381.423,E2 22381.423} C_VEL
LIN {X 0,Y 466.253,Z 886.862,A -85,B 0,C 180,E1 22379.308,E2 22379.308} C_VEL
LIN {X 0,Y 468.899,Z 869.231,A -85,B 0,C 180,E1 22377.21,E2 22377.21} C_VEL
LIN {X 0,Y 471.591,Z 851.473,A -85,B 0,C 180,E1 22375.379,E2 22375.379} C_VEL
LIN {X 0,Y 474.319,Z 832.149,A -85,B 0,C 180,E1 22373.681,E2 22373.681} C_VEL
LIN {X 0,Y 477.068,Z 812.005,A -85,B 0,C 180,E1 22372.169,E2 22372.169} C_VEL
LIN {X 0,Y 479.391,Z 792.696,A -85,B 0,C 180,E1 22370.964,E2 22370.964} C_VEL
LIN {X 0,Y 481.673,Z 771.956,A -85,B 0,C 180,E1 22369.874,E2 22369.874} C_VEL
LIN {X 0,Y 483.604,Z 749.854,A -85,B 0,C 180,E1 22368.958,E2 22368.958} C_VEL
LIN {X 0,Y 485.265,Z 726.88,A -85,B 0,C 180,E1 22368.227,E2 22368.227} C_VEL
LIN {X 0,Y 486.348,Z 704.887,A -85,B 0,C 180,E1 22367.739,E2 22367.739} C_VEL
LIN {X 0,Y 491.764,Z 496.733,A -85,B 0,C 180,E1 22364.156,E2 22364.156} C_VEL
LIN {X 0,Y 493.64,Z 424.701,A -85,B 0,C 180,E1 22362.888,E2 22362.888} C_VEL
LIN {X 0,Y 480.288,Z 405.683,A -85,B 0,C 180,E1 22360.702,E2 22360.702} C_VEL
LIN {X 0,Y 472.188,Z 394.922,A -85,B 0,C 180,E1 22359.282,E2 22359.282} C_VEL
LIN {X 0,Y 468.998,Z 390.642,A -85,B 0,C 180,E1 22358.696,E2 22358.696} C_VEL
LIN {X 0,Y 465.789,Z 386.278,A -85,B 0,C 180,E1 22358.089,E2 22358.089} C_VEL
LIN {X 0,Y 462.173,Z 381.978,A -85,B 0,C 180,E1 22357.4,E2 22357.4} C_VEL
LIN {X 0,Y 461.005,Z 380.064,A -85,B 0,C 180,E1 22357.159,E2 22357.159} C_VEL
LIN {X 0,Y 458.403,Z 377.671,A -85,B 0,C 180,E1 22356.662,E2 22356.662} C_VEL
LIN {X 0,Y 457.148,Z 374.655,A -85,B 0,C 180,E1 22356.37,E2 22356.37} C_VEL
LIN {X 0,Y 457.062,Z 374.103,A -85,B 0,C 180,E1 22356.313,E2 22356.313} C_VEL
LIN {X 0,Y 457.043,Z 374.109,A -85,B 0,C 180,E1 22352.631,E2 22352.631} C_VEL
LIN {X 0,Y 457.036,Z 374.08,A -85,B 0,C 180,E1 22348.913,E2 22348.913} C_VEL
LIN {X 0,Y 457.058,Z 374.099,A -85,B 0,C 180,E1 22345.251,E2 22345.251} C_VEL
LIN {X 0,Y 457.08,Z 374.098,A -85,B 0,C 180,E1 22341.562,E2 22341.562} C_VEL
LIN {X 0,Y 457.039,Z 374.078,A -85,B 0,C 180,E1 22337.91,E2 22337.91} C_VEL
LIN {X 0,Y 457.019,Z 374.117,A -85,B 0,C 180,E1 22334.285,E2 22334.285} C_VEL
LIN {X 0,Y 457.027,Z 374.12,A -85,B 0,C 180,E1 22330.59,E2 22330.59} C_VEL
LIN {X 0,Y 457.069,Z 374.111,A -85,B 0,C 180,E1 22327.037,E2 22327.037} C_VEL
LIN {X 0,Y 457.037,Z 374.114,A -85,B 0,C 180,E1 22323.387,E2 22323.387} C_VEL
LIN {X 0,Y 457.002,Z 374.118,A -85,B 0,C 180,E1 22319.875,E2 22319.875} C_VEL
LIN {X 0,Y 457.009,Z 374.12,A -85,B 0,C 180,E1 22316.237,E2 22316.237} C_VEL
LIN {X 0,Y 457.06,Z 374.111,A -85,B 0,C 180,E1 22312.711,E2 22312.711} C_VEL
LIN {X 0,Y 457.022,Z 374.117,A -85,B 0,C 180,E1 22309.028,E2 22309.028} C_VEL
LIN {X 0,Y 457.002,Z 374.121,A -85,B 0,C 180,E1 22305.428,E2 22305.428} C_VEL
LIN {X 0,Y 457.006,Z 374.083,A -85,B 0,C 180,E1 22301.699,E2 22301.699} C_VEL
LIN {X 0,Y 457.054,Z 374.106,A -85,B 0,C 180,E1 22298.168,E2 22298.168} C_VEL
LIN {X 0,Y 457.053,Z 374.104,A -85,B 0,C 180,E1 22294.472,E2 22294.472} C_VEL
LIN {X 0,Y 457.017,Z 374.084,A -85,B 0,C 180,E1 22290.943,E2 22290.943} C_VEL
LIN {X 0,Y 457.024,Z 374.1,A -85,B 0,C 180,E1 22287.291,E2 22287.291} C_VEL
LIN {X 0,Y 457.025,Z 374.093,A -85,B 0,C 180,E1 22285.257,E2 22285.257} C_VEL
LIN {X 0,Y 458.183,Z 377.348,A -85,B 0,C 180,E1 22284.67,E2 22284.67} C_VEL
LIN {X 0,Y 459.661,Z 379.348,A -85,B 0,C 180,E1 22284.188,E2 22284.188} C_VEL
LIN {X 0,Y 461.551,Z 383.197,A -85,B 0,C 180,E1 22283.436,E2 22283.436} C_VEL
LIN {X 0,Y 463.694,Z 387.194,A -85,B 0,C 180,E1 22282.706,E2 22282.706} C_VEL
LIN {X 0,Y 469.674,Z 395.527,A -85,B 0,C 180,E1 22281.566,E2 22281.566} C_VEL
LIN {X 0,Y 478.637,Z 408.263,A -85,B 0,C 180,E1 22279.954,E2 22279.954} C_VEL
LIN {X 0,Y 489.814,Z 425.456,A -85,B 0,C 180,E1 22278.067,E2 22278.067} C_VEL
LIN {X 0,Y 493.945,Z 432.336,A -85,B 0,C 180,E1 22277.396,E2 22277.396} C_VEL
LIN {X 0,Y 488.384,Z 644.564,A -85,B 0,C 180,E1 22273.729,E2 22273.729} C_VEL
LIN {X 0,Y 485.879,Z 739.504,A -85,B 0,C 180,E1 22272.09,E2 22272.09} C_VEL
LIN {X 0,Y 484.467,Z 762.623,A -85,B 0,C 180,E1 22271.504,E2 22271.504} C_VEL
LIN {X 0,Y 482.794,Z 784.49,A -85,B 0,C 180,E1 22270.754,E2 22270.754} C_VEL
LIN {X 0,Y 480.766,Z 805.312,A -85,B 0,C 180,E1 22269.828,E2 22269.828} C_VEL
LIN {X 0,Y 478.544,Z 825.655,A -85,B 0,C 180,E1 22268.734,E2 22268.734} C_VEL
LIN {X 0,Y 475.969,Z 846.468,A -85,B 0,C 180,E1 22267.375,E2 22267.375} C_VEL
LIN {X 0,Y 473.319,Z 867.073,A -85,B 0,C 180,E1 22265.79,E2 22265.79} C_VEL
LIN {X 0,Y 470.605,Z 886.213,A -85,B 0,C 180,E1 22264.045,E2 22264.045} C_VEL
LIN {X 0,Y 467.948,Z 905.11,A -85,B 0,C 180,E1 22262.056,E2 22262.056} C_VEL
LIN {X 0,Y 465.846,Z 919.625,A -85,B 0,C 180,E1 22260.287,E2 22260.287} C_VEL
LIN {X 0,Y 463.538,Z 935.77,A -85,B 0,C 180,E1 22258.046,E2 22258.046} C_VEL
LIN {X 0,Y 461.522,Z 950.436,A -85,B 0,C 180,E1 22255.674,E2 22255.674} C_VEL
LIN {X 0,Y 459.757,Z 964.548,A -85,B 0,C 180,E1 22253.043,E2 22253.043} C_VEL
LIN {X 0,Y 458.46,Z 976.017,A -85,B 0,C 180,E1 22250.554,E2 22250.554} C_VEL
LIN {X 0,Y 457.389,Z 987.232,A -85,B 0,C 180,E1 22247.688,E2 22247.688} C_VEL
LIN {X 0,Y 456.714,Z 996.178,A -85,B 0,C 180,E1 22244.97,E2 22244.97} C_VEL
LIN {X 0,Y 456.267,Z 1003.655,A -85,B 0,C 180,E1 22242.143,E2 22242.143} C_VEL
LIN {X 0,Y 456.04,Z 1009.599,A -85,B 0,C 180,E1 22239.336,E2 22239.336} C_VEL
LIN {X 0,Y 455.942,Z 1013.8,A -85,B 0,C 180,E1 22236.547,E2 22236.547} C_VEL
LIN {X 0,Y 455.904,Z 1016.655,A -85,B 0,C 180,E1 22233.743,E2 22233.743} C_VEL
LIN {X 0,Y 455.893,Z 1017.826,A -85,B 0,C 180,E1 22231.006,E2 22231.006} C_VEL
LIN {X 0,Y 455.908,Z 1017.736,A -85,B 0,C 180,E1 22228.492,E2 22228.492} C_VEL
LIN {X 0,Y 455.909,Z 1016.069,A -85,B 0,C 180,E1 22225.599,E2 22225.599} C_VEL
LIN {X 0,Y 455.93,Z 1013.321,A -85,B 0,C 180,E1 22223.074,E2 22223.074} C_VEL
LIN {X 0,Y 456.047,Z 1008.593,A -85,B 0,C 180,E1 22220.155,E2 22220.155} C_VEL
LIN {X 0,Y 456.297,Z 1003.049,A -85,B 0,C 180,E1 22217.601,E2 22217.601} C_VEL
LIN {X 0,Y 456.792,Z 994.964,A -85,B 0,C 180,E1 22214.644,E2 22214.644} C_VEL
LIN {X 0,Y 457.471,Z 986.321,A -85,B 0,C 180,E1 22212.053,E2 22212.053} C_VEL
LIN {X 0,Y 458.571,Z 974.878,A -85,B 0,C 180,E1 22209.185,E2 22209.185} C_VEL
LIN {X 0,Y 460.021,Z 962.427,A -85,B 0,C 180,E1 22206.522,E2 22206.522} C_VEL
LIN {X 0,Y 461.836,Z 948.129,A -85,B 0,C 180,E1 22203.932,E2 22203.932} C_VEL
LIN {X 0,Y 464.104,Z 931.668,A -85,B 0,C 180,E1 22201.361,E2 22201.361} C_VEL
LIN {X 0,Y 466.448,Z 915.578,A -85,B 0,C 180,E1 22199.186,E2 22199.186} C_VEL
LIN {X 0,Y 468.971,Z 897.791,A -85,B 0,C 180,E1 22197.141,E2 22197.141} C_VEL
LIN {X 0,Y 471.688,Z 878.773,A -85,B 0,C 180,E1 22195.24,E2 22195.24} C_VEL
LIN {X 0,Y 474.29,Z 859.382,A -85,B 0,C 180,E1 22193.592,E2 22193.592} C_VEL
LIN {X 0,Y 477.079,Z 837.915,A -85,B 0,C 180,E1 22192.038,E2 22192.038} C_VEL
LIN {X 0,Y 479.31,Z 818.838,A -85,B 0,C 180,E1 22190.88,E2 22190.88} C_VEL
LIN {X 0,Y 481.629,Z 796.529,A -85,B 0,C 180,E1 22189.754,E2 22189.754} C_VEL
LIN {X 0,Y 483.525,Z 775.138,A -85,B 0,C 180,E1 22188.901,E2 22188.901} C_VEL
LIN {X 0,Y 485.218,Z 751.512,A -85,B 0,C 180,E1 22188.19,E2 22188.19} C_VEL
LIN {X 0,Y 486.259,Z 729.771,A -85,B 0,C 180,E1 22187.725,E2 22187.725} C_VEL
LIN {X 0,Y 491.502,Z 522.39,A -85,B 0,C 180,E1 22184.169,E2 22184.169} C_VEL
LIN {X 0,Y 493.808,Z 431.739,A -85,B 0,C 180,E1 22182.575,E2 22182.575} C_VEL
LIN {X 0,Y 480.763,Z 411.392,A -85,B 0,C 180,E1 22180.417,E2 22180.417} C_VEL
LIN {X 0,Y 470.342,Z 396.471,A -85,B 0,C 180,E1 22178.564,E2 22178.564} C_VEL
LIN {X 0,Y 466.772,Z 391.526,A -85,B 0,C 180,E1 22177.896,E2 22177.896} C_VEL
LIN {X 0,Y 463.137,Z 386.454,A -85,B 0,C 180,E1 22177.191,E2 22177.191} C_VEL
LIN {X 0,Y 461.228,Z 382.762,A -85,B 0,C 180,E1 22176.471,E2 22176.471} C_VEL
LIN {X 0,Y 459.304,Z 378.736,A -85,B 0,C 180,E1 22175.69,E2 22175.69} C_VEL
LIN {X 0,Y 457.538,Z 376.086,A -85,B 0,C 180,E1 22175.081,E2 22175.081} C_VEL
LIN {X 0,Y 457.024,Z 374.088,A -85,B 0,C 180,E1 22174.744,E2 22174.744} C_VEL
LIN {X 0,Y 457.023,Z 374.109,A -85,B 0,C 180,E1 22171.085,E2 22171.085} C_VEL
LIN {X 0,Y 457.064,Z 374.094,A -85,B 0,C 180,E1 22167.63,E2 22167.63} C_VEL
LIN {X 0,Y 457.04,Z 374.074,A -85,B 0,C 180,E1 22164.01,E2 22164.01} C_VEL
LIN {X 0,Y 457.01,Z 374.117,A -85,B 0,C 180,E1 22160.49,E2 22160.49} C_VEL
LIN {X 0,Y 457.006,Z 374.081,A -85,B 0,C 180,E1 22156.785,E2 22156.785} C_VEL
LIN {X 0,Y 457.05,Z 374.109,A -85,B 0,C 180,E1 22153.25,E2 22153.25} C_VEL
LIN {X 0,Y 457.032,Z 374.111,A -85,B 0,C 180,E1 22149.571,E2 22149.571} C_VEL
LIN {X 0,Y 456.991,Z 374.116,A -85,B 0,C 180,E1 22146.154,E2 22146.154} C_VEL
LIN {X 0,Y 457.006,Z 374.111,A -85,B 0,C 180,E1 22142.508,E2 22142.508} C_VEL
LIN {X 0,Y 457.062,Z 374.106,A -85,B 0,C 180,E1 22138.997,E2 22138.997} C_VEL
LIN {X 0,Y 457.026,Z 374.113,A -85,B 0,C 180,E1 22135.357,E2 22135.357} C_VEL
LIN {X 0,Y 457.008,Z 374.116,A -85,B 0,C 180,E1 22131.824,E2 22131.824} C_VEL
LIN {X 0,Y 457.034,Z 374.108,A -85,B 0,C 180,E1 22128.261,E2 22128.261} C_VEL
LIN {X 0,Y 457.076,Z 374.099,A -85,B 0,C 180,E1 22124.651,E2 22124.651} C_VEL
LIN {X 0,Y 457.047,Z 374.094,A -85,B 0,C 180,E1 22120.9,E2 22120.9} C_VEL
LIN {X 0,Y 457.021,Z 374.09,A -85,B 0,C 180,E1 22117.353,E2 22117.353} C_VEL
LIN {X 0,Y 457.036,Z 374.117,A -85,B 0,C 180,E1 22113.634,E2 22113.634} C_VEL
LIN {X 0,Y 457.073,Z 374.076,A -85,B 0,C 180,E1 22110.015,E2 22110.015} C_VEL
LIN {X 0,Y 457.066,Z 374.088,A -85,B 0,C 180,E1 22106.396,E2 22106.396} C_VEL
LIN {X 0,Y 457.079,Z 374.29,A -85,B 0,C 180,E1 22103.552,E2 22103.552} C_VEL
LIN {X 0,Y 458.203,Z 377.375,A -85,B 0,C 180,E1 22103.28,E2 22103.28} C_VEL
LIN {X 0,Y 460.647,Z 379.853,A -85,B 0,C 180,E1 22102.807,E2 22102.807} C_VEL
LIN {X 0,Y 461.539,Z 380.728,A -85,B 0,C 180,E1 22102.638,E2 22102.638} C_VEL
LIN {X 0,Y 464.119,Z 384.59,A -85,B 0,C 180,E1 22102.122,E2 22102.122} C_VEL
LIN {X 0,Y 465.985,Z 386.659,A -85,B 0,C 180,E1 22101.774,E2 22101.774} C_VEL
LIN {X 0,Y 469.36,Z 390.996,A -85,B 0,C 180,E1 22101.144,E2 22101.144} C_VEL
LIN {X 0,Y 481.601,Z 407.538,A -85,B 0,C 180,E1 22098.981,E2 22098.981} C_VEL
LIN {X 0,Y 493.723,Z 424.857,A -85,B 0,C 180,E1 22097.008,E2 22097.008} C_VEL
LIN {X 0,Y 489.144,Z 596.368,A -85,B 0,C 180,E1 22094.033,E2 22094.033} C_VEL
LIN {X 0,Y 488.232,Z 604.069,A -85,B 0,C 180,E1 22093.983,E2 22093.983} C_VEL
LIN {X 0,Y 483.201,Z 624.67,A -85,B 0,C 180,E1 22094.146,E2 22094.146} C_VEL
LIN {X 0,Y 482.486,Z 631.277,A -85,B 0,C 180,E1 22094.094,E2 22094.094} C_VEL
LIN {X 0,Y 480.13,Z 713.246,A -85,B 0,C 180,E1 22092.656,E2 22092.656} C_VEL
LIN {X 0,Y 478.736,Z 735.607,A -85,B 0,C 180,E1 22092.073,E2 22092.073} C_VEL
LIN {X 0,Y 477.005,Z 757.262,A -85,B 0,C 180,E1 22091.315,E2 22091.315} C_VEL
LIN {X 0,Y 474.752,Z 778.988,A -85,B 0,C 180,E1 22090.324,E2 22090.324} C_VEL
LIN {X 0,Y 472.342,Z 799.547,A -85,B 0,C 180,E1 22089.182,E2 22089.182} C_VEL
LIN {X 0,Y 469.604,Z 819.667,A -85,B 0,C 180,E1 22087.815,E2 22087.815} C_VEL
LIN {X 0,Y 466.772,Z 839.413,A -85,B 0,C 180,E1 22086.238,E2 22086.238} C_VEL
LIN {X 0,Y 463.911,Z 857.577,A -85,B 0,C 180,E1 22084.525,E2 22084.525} C_VEL
LIN {X 0,Y 461.001,Z 875.808,A -85,B 0,C 180,E1 22082.535,E2 22082.535} C_VEL
LIN {X 0,Y 458.413,Z 891.767,A -85,B 0,C 180,E1 22080.509,E2 22080.509} C_VEL
LIN {X 0,Y 455.586,Z 909.731,A -85,B 0,C 180,E1 22077.866,E2 22077.866} C_VEL
LIN {X 0,Y 453.534,Z 924.024,A -85,B 0,C 180,E1 22075.457,E2 22075.457} C_VEL
LIN {X 0,Y 451.8,Z 936.884,A -85,B 0,C 180,E1 22072.92,E2 22072.92} C_VEL
LIN {X 0,Y 450.346,Z 949.266,A -85,B 0,C 180,E1 22070.091,E2 22070.091} C_VEL
LIN {X 0,Y 449.376,Z 958.917,A -85,B 0,C 180,E1 22067.478,E2 22067.478} C_VEL
LIN {X 0,Y 448.623,Z 968.229,A -85,B 0,C 180,E1 22064.453,E2 22064.453} C_VEL
LIN {X 0,Y 448.246,Z 974.763,A -85,B 0,C 180,E1 22061.84,E2 22061.84} C_VEL
LIN {X 0,Y 448.024,Z 980.566,A -85,B 0,C 180,E1 22058.857,E2 22058.857} C_VEL
LIN {X 0,Y 447.94,Z 984.223,A -85,B 0,C 180,E1 22056.278,E2 22056.278} C_VEL
LIN {X 0,Y 447.888,Z 986.893,A -85,B 0,C 180,E1 22053.327,E2 22053.327} C_VEL
LIN {X 0,Y 447.888,Z 987.864,A -85,B 0,C 180,E1 22050.767,E2 22050.767} C_VEL
LIN {X 0,Y 447.911,Z 987.618,A -85,B 0,C 180,E1 22047.953,E2 22047.953} C_VEL
LIN {X 0,Y 447.906,Z 985.882,A -85,B 0,C 180,E1 22045.262,E2 22045.262} C_VEL
LIN {X 0,Y 447.94,Z 982.897,A -85,B 0,C 180,E1 22042.562,E2 22042.562} C_VEL
LIN {X 0,Y 448.082,Z 978.171,A -85,B 0,C 180,E1 22039.718,E2 22039.718} C_VEL
LIN {X 0,Y 448.392,Z 972.242,A -85,B 0,C 180,E1 22036.985,E2 22036.985} C_VEL
LIN {X 0,Y 448.926,Z 964.289,A -85,B 0,C 180,E1 22034.102,E2 22034.102} C_VEL
LIN {X 0,Y 449.776,Z 954.847,A -85,B 0,C 180,E1 22031.263,E2 22031.263} C_VEL
LIN {X 0,Y 450.94,Z 943.911,A -85,B 0,C 180,E1 22028.542,E2 22028.542} C_VEL
LIN {X 0,Y 452.519,Z 931.402,A -85,B 0,C 180,E1 22025.859,E2 22025.859} C_VEL
LIN {X 0,Y 454.323,Z 918.369,A -85,B 0,C 180,E1 22023.467,E2 22023.467} C_VEL
LIN {X 0,Y 456.778,Z 901.982,A -85,B 0,C 180,E1 22020.855,E2 22020.855} C_VEL
LIN {X 0,Y 459.233,Z 886.678,A -85,B 0,C 180,E1 22018.72,E2 22018.72} C_VEL
LIN {X 0,Y 462.093,Z 868.992,A -85,B 0,C 180,E1 22016.598,E2 22016.598} C_VEL
LIN {X 0,Y 464.971,Z 851.113,A -85,B 0,C 180,E1 22014.738,E2 22014.738} C_VEL
LIN {X 0,Y 467.881,Z 831.643,A -85,B 0,C 180,E1 22013.023,E2 22013.023} C_VEL
LIN {X 0,Y 470.759,Z 811.653,A -85,B 0,C 180,E1 22011.52,E2 22011.52} C_VEL
LIN {X 0,Y 473.268,Z 791.863,A -85,B 0,C 180,E1 22010.282,E2 22010.282} C_VEL
LIN {X 0,Y 475.671,Z 770.673,A -85,B 0,C 180,E1 22009.176,E2 22009.176} C_VEL
LIN {X 0,Y 477.648,Z 749.185,A -85,B 0,C 180,E1 22008.288,E2 22008.288} C_VEL
LIN {X 0,Y 479.464,Z 724.79,A -85,B 0,C 180,E1 22007.531,E2 22007.531} C_VEL
LIN {X 0,Y 480.539,Z 703.135,A -85,B 0,C 180,E1 22007.058,E2 22007.058} C_VEL
LIN {X 0,Y 486.32,Z 493.529,A -85,B 0,C 180,E1 22003.419,E2 22003.419} C_VEL
LIN {X 0,Y 488.132,Z 428.652,A -85,B 0,C 180,E1 22002.266,E2 22002.266} C_VEL
LIN {X 0,Y 476.189,Z 411.532,A -85,B 0,C 180,E1 22000.255,E2 22000.255} C_VEL
LIN {X 0,Y 465.577,Z 397.233,A -85,B 0,C 180,E1 21998.324,E2 21998.324} C_VEL
LIN {X 0,Y 461.09,Z 391.532,A -85,B 0,C 180,E1 21997.464,E2 21997.464} C_VEL
LIN {X 0,Y 457.369,Z 386.662,A -85,B 0,C 180,E1 21996.72,E2 21996.72} C_VEL
LIN {X 0,Y 454.458,Z 383.266,A -85,B 0,C 180,E1 21996.131,E2 21996.131} C_VEL
LIN {X 0,Y 453.213,Z 381.097,A -85,B 0,C 180,E1 21995.855,E2 21995.855} C_VEL
LIN {X 0,Y 450.429,Z 378.573,A -85,B 0,C 180,E1 21995.289,E2 21995.289} C_VEL
LIN {X 0,Y 449.165,Z 375.499,A -85,B 0,C 180,E1 21994.974,E2 21994.974} C_VEL
LIN {X 0,Y 449.099,Z 375.067,A -85,B 0,C 180,E1 21994.902,E2 21994.902} C_VEL
LIN {X 0,Y 449.115,Z 375.094,A -85,B 0,C 180,E1 21991.247,E2 21991.247} C_VEL
LIN {X 0,Y 449.138,Z 375.086,A -85,B 0,C 180,E1 21987.584,E2 21987.584} C_VEL
LIN {X 0,Y 449.118,Z 375.061,A -85,B 0,C 180,E1 21983.903,E2 21983.903} C_VEL
LIN {X 0,Y 449.091,Z 375.107,A -85,B 0,C 180,E1 21980.324,E2 21980.324} C_VEL
LIN {X 0,Y 449.081,Z 375.062,A -85,B 0,C 180,E1 21976.558,E2 21976.558} C_VEL
LIN {X 0,Y 449.115,Z 375.1,A -85,B 0,C 180,E1 21972.995,E2 21972.995} C_VEL
LIN {X 0,Y 449.129,Z 375.097,A -85,B 0,C 180,E1 21969.224,E2 21969.224} C_VEL
LIN {X 0,Y 449.086,Z 375.104,A -85,B 0,C 180,E1 21965.622,E2 21965.622} C_VEL
LIN {X 0,Y 449.067,Z 375.105,A -85,B 0,C 180,E1 21962.042,E2 21962.042} C_VEL
LIN {X 0,Y 449.085,Z 375.101,A -85,B 0,C 180,E1 21958.469,E2 21958.469} C_VEL
LIN {X 0,Y 449.112,Z 375.097,A -85,B 0,C 180,E1 21954.763,E2 21954.763} C_VEL
LIN {X 0,Y 449.073,Z 375.103,A -85,B 0,C 180,E1 21951.163,E2 21951.163} C_VEL
LIN {X 0,Y 449.058,Z 375.103,A -85,B 0,C 180,E1 21947.527,E2 21947.527} C_VEL
LIN {X 0,Y 449.069,Z 375.089,A -85,B 0,C 180,E1 21943.841,E2 21943.841} C_VEL
LIN {X 0,Y 449.112,Z 375.093,A -85,B 0,C 180,E1 21940.221,E2 21940.221} C_VEL
LIN {X 0,Y 449.1,Z 375.068,A -85,B 0,C 180,E1 21936.654,E2 21936.654} C_VEL
LIN {X 0,Y 449.078,Z 375.11,A -85,B 0,C 180,E1 21933.13,E2 21933.13} C_VEL
LIN {X 0,Y 449.083,Z 375.088,A -85,B 0,C 180,E1 21929.346,E2 21929.346} C_VEL
LIN {X 0,Y 449.123,Z 375.251,A -85,B 0,C 180,E1 21926.527,E2 21926.527} C_VEL
LIN {X 0,Y 450.523,Z 378.692,A -85,B 0,C 180,E1 21925.842,E2 21925.842} C_VEL
LIN {X 0,Y 451.745,Z 380.408,A -85,B 0,C 180,E1 21925.413,E2 21925.413} C_VEL
LIN {X 0,Y 453.778,Z 384.341,A -85,B 0,C 180,E1 21924.585,E2 21924.585} C_VEL
LIN {X 0,Y 455.178,Z 386.938,A -85,B 0,C 180,E1 21924.13,E2 21924.13} C_VEL
LIN {X 0,Y 465.096,Z 400.339,A -85,B 0,C 180,E1 21922.158,E2 21922.158} C_VEL
LIN {X 0,Y 477.654,Z 418.723,A -85,B 0,C 180,E1 21919.855,E2 21919.855} C_VEL
LIN {X 0,Y 488.416,Z 435.73,A -85,B 0,C 180,E1 21918.027,E2 21918.027} C_VEL
LIN {X 0,Y 482.516,Z 647.408,A -85,B 0,C 180,E1 21914.336,E2 21914.336} C_VEL
LIN {X 0,Y 479.934,Z 739.31,A -85,B 0,C 180,E1 21912.732,E2 21912.732} C_VEL
LIN {X 0,Y 478.428,Z 762.451,A -85,B 0,C 180,E1 21912.142,E2 21912.142} C_VEL
LIN {X 0,Y 476.599,Z 785.029,A -85,B 0,C 180,E1 21911.359,E2 21911.359} C_VEL
LIN {X 0,Y 474.382,Z 806.299,A -85,B 0,C 180,E1 21910.395,E2 21910.395} C_VEL
LIN {X 0,Y 471.904,Z 827.556,A -85,B 0,C 180,E1 21909.226,E2 21909.226} C_VEL
LIN {X 0,Y 469.101,Z 848.623,A -85,B 0,C 180,E1 21907.809,E2 21907.809} C_VEL
LIN {X 0,Y 466.054,Z 870.323,A -85,B 0,C 180,E1 21906.071,E2 21906.071} C_VEL
LIN {X 0,Y 463.313,Z 888.648,A -85,B 0,C 180,E1 21904.352,E2 21904.352} C_VEL
LIN {X 0,Y 460.441,Z 907.526,A -85,B 0,C 180,E1 21902.285,E2 21902.285} C_VEL
LIN {X 0,Y 457.879,Z 924.552,A -85,B 0,C 180,E1 21900.145,E2 21900.145} C_VEL
LIN {X 0,Y 455.672,Z 939.149,A -85,B 0,C 180,E1 21898.003,E2 21898.003} C_VEL
LIN {X 0,Y 453.606,Z 953.516,A -85,B 0,C 180,E1 21895.594,E2 21895.594} C_VEL
LIN {X 0,Y 451.772,Z 967.086,A -85,B 0,C 180,E1 21892.922,E2 21892.922} C_VEL
LIN {X 0,Y 450.32,Z 979.465,A -85,B 0,C 180,E1 21890.084,E2 21890.084} C_VEL
LIN {X 0,Y 449.363,Z 989.066,A -85,B 0,C 180,E1 21887.479,E2 21887.479} C_VEL
LIN {X 0,Y 448.615,Z 998.349,A -85,B 0,C 180,E1 21884.454,E2 21884.454} C_VEL
LIN {X 0,Y 448.238,Z 1004.866,A -85,B 0,C 180,E1 21881.841,E2 21881.841} C_VEL
LIN {X 0,Y 448.02,Z 1010.637,A -85,B 0,C 180,E1 21878.857,E2 21878.857} C_VEL
LIN {X 0,Y 447.935,Z 1014.439,A -85,B 0,C 180,E1 21876.15,E2 21876.15} C_VEL
LIN {X 0,Y 447.886,Z 1016.985,A -85,B 0,C 180,E1 21873.199,E2 21873.199} C_VEL
LIN {X 0,Y 447.885,Z 1017.871,A -85,B 0,C 180,E1 21870.768,E2 21870.768} C_VEL
LIN {X 0,Y 447.912,Z 1017.595,A -85,B 0,C 180,E1 21867.954,E2 21867.954} C_VEL
LIN {X 0,Y 447.909,Z 1015.842,A -85,B 0,C 180,E1 21865.263,E2 21865.263} C_VEL
LIN {X 0,Y 447.953,Z 1012.682,A -85,B 0,C 180,E1 21862.434,E2 21862.434} C_VEL
LIN {X 0,Y 448.102,Z 1007.83,A -85,B 0,C 180,E1 21859.589,E2 21859.589} C_VEL
LIN {X 0,Y 448.438,Z 1001.522,A -85,B 0,C 180,E1 21856.725,E2 21856.725} C_VEL
LIN {X 0,Y 448.966,Z 993.749,A -85,B 0,C 180,E1 21853.972,E2 21853.972} C_VEL
LIN {X 0,Y 449.819,Z 984.451,A -85,B 0,C 180,E1 21851.2,E2 21851.2} C_VEL
LIN {X 0,Y 450.964,Z 973.729,A -85,B 0,C 180,E1 21848.544,E2 21848.544} C_VEL
LIN {X 0,Y 452.556,Z 961.104,A -85,B 0,C 180,E1 21845.847,E2 21845.847} C_VEL
LIN {X 0,Y 454.47,Z 947.357,A -85,B 0,C 180,E1 21843.336,E2 21843.336} C_VEL
LIN {X 0,Y 456.826,Z 931.52,A -85,B 0,C 180,E1 21840.843,E2 21840.843} C_VEL
LIN {X 0,Y 459.268,Z 915.298,A -85,B 0,C 180,E1 21838.651,E2 21838.651} C_VEL
LIN {X 0,Y 461.978,Z 897.462,A -85,B 0,C 180,E1 21836.577,E2 21836.577} C_VEL
LIN {X 0,Y 464.861,Z 878.46,A -85,B 0,C 180,E1 21834.654,E2 21834.654} C_VEL
LIN {X 0,Y 467.635,Z 859.2,A -85,B 0,C 180,E1 21833.001,E2 21833.001} C_VEL
LIN {X 0,Y 470.476,Z 838.721,A -85,B 0,C 180,E1 21831.493,E2 21831.493} C_VEL
LIN {X 0,Y 472.974,Z 818.53,A -85,B 0,C 180,E1 21830.253,E2 21830.253} C_VEL
LIN {X 0,Y 475.439,Z 796.223,A -85,B 0,C 180,E1 21829.119,E2 21829.119} C_VEL
LIN {X 0,Y 477.445,Z 774.944,A -85,B 0,C 180,E1 21828.266,E2 21828.266} C_VEL
LIN {X 0,Y 479.231,Z 751.373,A -85,B 0,C 180,E1 21827.552,E2 21827.552} C_VEL
LIN {X 0,Y 480.325,Z 729.684,A -85,B 0,C 180,E1 21827.083,E2 21827.083} C_VEL
LIN {X 0,Y 485.9,Z 522.839,A -85,B 0,C 180,E1 21823.501,E2 21823.501} C_VEL
LIN {X 0,Y 488.256,Z 435.364,A -85,B 0,C 180,E1 21821.946,E2 21821.946} C_VEL
LIN {X 0,Y 476.292,Z 416.704,A -85,B 0,C 180,E1 21819.91,E2 21819.91} C_VEL
LIN {X 0,Y 466.35,Z 402.289,A -85,B 0,C 180,E1 21818.092,E2 21818.092} C_VEL
LIN {X 0,Y 457.247,Z 389.598,A -85,B 0,C 180,E1 21816.302,E2 21816.302} C_VEL
LIN {X 0,Y 454.406,Z 385.499,A -85,B 0,C 180,E1 21815.668,E2 21815.668} C_VEL
LIN {X 0,Y 451.849,Z 380.753,A -85,B 0,C 180,E1 21814.659,E2 21814.659} C_VEL
LIN {X 0,Y 449.339,Z 376.207,A -85,B 0,C 180,E1 21813.646,E2 21813.646} C_VEL
LIN {X 0,Y 449.096,Z 375.074,A -85,B 0,C 180,E1 21813.406,E2 21813.406} C_VEL
LIN {X 0,Y 449.134,Z 375.062,A -85,B 0,C 180,E1 21809.76,E2 21809.76} C_VEL
LIN {X 0,Y 449.113,Z 375.097,A -85,B 0,C 180,E1 21806.013,E2 21806.013} C_VEL
LIN {X 0,Y 449.073,Z 375.077,A -85,B 0,C 180,E1 21802.379,E2 21802.379} C_VEL
LIN {X 0,Y 449.066,Z 375.074,A -85,B 0,C 180,E1 21798.7,E2 21798.7} C_VEL
LIN {X 0,Y 449.094,Z 375.098,A -85,B 0,C 180,E1 21795.099,E2 21795.099} C_VEL
LIN {X 0,Y 449.112,Z 375.1,A -85,B 0,C 180,E1 21791.428,E2 21791.428} C_VEL
LIN {X 0,Y 449.069,Z 375.107,A -85,B 0,C 180,E1 21787.806,E2 21787.806} C_VEL
LIN {X 0,Y 449.055,Z 375.11,A -85,B 0,C 180,E1 21784.142,E2 21784.142} C_VEL
LIN {X 0,Y 449.074,Z 375.11,A -85,B 0,C 180,E1 21780.51,E2 21780.51} C_VEL
LIN {X 0,Y 449.116,Z 375.104,A -85,B 0,C 180,E1 21776.937,E2 21776.937} C_VEL
LIN {X 0,Y 449.097,Z 375.105,A -85,B 0,C 180,E1 21773.223,E2 21773.223} C_VEL
LIN {X 0,Y 449.074,Z 375.108,A -85,B 0,C 180,E1 21769.61,E2 21769.61} C_VEL
LIN {X 0,Y 449.08,Z 375.108,A -85,B 0,C 180,E1 21765.823,E2 21765.823} C_VEL
LIN {X 0,Y 449.109,Z 375.058,A -85,B 0,C 180,E1 21762.241,E2 21762.241} C_VEL
LIN {X 0,Y 449.139,Z 375.094,A -85,B 0,C 180,E1 21758.501,E2 21758.501} C_VEL
LIN {X 0,Y 449.104,Z 375.076,A -85,B 0,C 180,E1 21754.835,E2 21754.835} C_VEL
LIN {X 0,Y 449.089,Z 375.073,A -85,B 0,C 180,E1 21751.255,E2 21751.255} C_VEL
LIN {X 0,Y 449.108,Z 375.105,A -85,B 0,C 180,E1 21747.551,E2 21747.551} C_VEL
LIN {X 0,Y 449.128,Z 375.309,A -85,B 0,C 180,E1 21744.935,E2 21744.935} C_VEL
LIN {X 0,Y 450.228,Z 378.268,A -85,B 0,C 180,E1 21744.654,E2 21744.654} C_VEL
LIN {X 0,Y 452.858,Z 380.886,A -85,B 0,C 180,E1 21744.112,E2 21744.112} C_VEL
LIN {X 0,Y 453.712,Z 381.827,A -85,B 0,C 180,E1 21743.937,E2 21743.937} C_VEL
LIN {X 0,Y 456.206,Z 385.605,A -85,B 0,C 180,E1 21743.406,E2 21743.406} C_VEL
LIN {X 0,Y 458.364,Z 387.862,A -85,B 0,C 180,E1 21742.983,E2 21742.983} C_VEL
LIN {X 0,Y 461.712,Z 392.147,A -85,B 0,C 180,E1 21742.322,E2 21742.322} C_VEL
LIN {X 0,Y 471.046,Z 404.589,A -85,B 0,C 180,E1 21740.565,E2 21740.565} C_VEL
LIN {X 0,Y 481.881,Z 419.556,A -85,B 0,C 180,E1 21738.674,E2 21738.674} C_VEL
LIN {X 0,Y 488.188,Z 429.021,A -85,B 0,C 180,E1 21737.627,E2 21737.627} C_VEL
LIN {X 0,Y 482.548,Z 628.96,A -85,B 0,C 180,E1 21734.135,E2 21734.135} C_VEL
LIN {X 0,Y 482.486,Z 631.277,A -85,B 0,C 180,E1 21734.094,E2 21734.094} C_VEL
LIN {X 0,Y 481.562,Z 638.978,A -85,B 0,C 180,E1 21734.045,E2 21734.045} C_VEL
LIN {X 0,Y 476.504,Z 659.572,A -85,B 0,C 180,E1 21734.214,E2 21734.214} C_VEL
LIN {X 0,Y 475.797,Z 666.177,A -85,B 0,C 180,E1 21734.161,E2 21734.161} C_VEL
LIN {X 0,Y 474.209,Z 715.308,A -85,B 0,C 180,E1 21733.275,E2 21733.275} C_VEL
LIN {X 0,Y 472.738,Z 736.97,A -85,B 0,C 180,E1 21732.691,E2 21732.691} C_VEL
LIN {X 0,Y 470.844,Z 759.179,A -85,B 0,C 180,E1 21731.895,E2 21731.895} C_VEL
LIN {X 0,Y 468.543,Z 780.068,A -85,B 0,C 180,E1 21730.923,E2 21730.923} C_VEL
LIN {X 0,Y 465.945,Z 800.876,A -85,B 0,C 180,E1 21729.746,E2 21729.746} C_VEL
LIN {X 0,Y 463.085,Z 820.785,A -85,B 0,C 180,E1 21728.373,E2 21728.373} C_VEL
LIN {X 0,Y 459.955,Z 841.181,A -85,B 0,C 180,E1 21726.707,E2 21726.707} C_VEL
LIN {X 0,Y 457.069,Z 858.552,A -85,B 0,C 180,E1 21725.041,E2 21725.041} C_VEL
LIN {X 0,Y 453.823,Z 877.532,A -85,B 0,C 180,E1 21722.921,E2 21722.921} C_VEL
LIN {X 0,Y 451.105,Z 893.368,A -85,B 0,C 180,E1 21720.867,E2 21720.867} C_VEL
LIN {X 0,Y 448.4,Z 909.134,A -85,B 0,C 180,E1 21718.498,E2 21718.498} C_VEL
LIN {X 0,Y 446.027,Z 924.03,A -85,B 0,C 180,E1 21715.917,E2 21715.917} C_VEL
LIN {X 0,Y 444.126,Z 937.12,A -85,B 0,C 180,E1 21713.288,E2 21713.288} C_VEL
LIN {X 0,Y 442.597,Z 949.136,A -85,B 0,C 180,E1 21710.494,E2 21710.494} C_VEL
LIN {X 0,Y 441.523,Z 958.918,A -85,B 0,C 180,E1 21707.799,E2 21707.799} C_VEL
LIN {X 0,Y 440.703,Z 968.231,A -85,B 0,C 180,E1 21704.718,E2 21704.718} C_VEL
LIN {X 0,Y 440.286,Z 974.764,A -85,B 0,C 180,E1 21702.058,E2 21702.058} C_VEL
LIN {X 0,Y 440.037,Z 980.567,A -85,B 0,C 180,E1 21699.019,E2 21699.019} C_VEL
LIN {X 0,Y 439.946,Z 984.224,A -85,B 0,C 180,E1 21696.393,E2 21696.393} C_VEL
LIN {X 0,Y 439.89,Z 986.893,A -85,B 0,C 180,E1 21693.387,E2 21693.387} C_VEL
LIN {X 0,Y 439.889,Z 987.864,A -85,B 0,C 180,E1 21690.781,E2 21690.781} C_VEL
LIN {X 0,Y 439.912,Z 987.618,A -85,B 0,C 180,E1 21687.916,E2 21687.916} C_VEL
LIN {X 0,Y 439.908,Z 985.881,A -85,B 0,C 180,E1 21685.176,E2 21685.176} C_VEL
LIN {X 0,Y 439.951,Z 982.896,A -85,B 0,C 180,E1 21682.426,E2 21682.426} C_VEL
LIN {X 0,Y 440.11,Z 978.17,A -85,B 0,C 180,E1 21679.529,E2 21679.529} C_VEL
LIN {X 0,Y 440.442,Z 972.241,A -85,B 0,C 180,E1 21676.746,E2 21676.746} C_VEL
LIN {X 0,Y 441.023,Z 964.286,A -85,B 0,C 180,E1 21673.81,E2 21673.81} C_VEL
LIN {X 0,Y 441.928,Z 955.082,A -85,B 0,C 180,E1 21670.988,E2 21670.988} C_VEL
LIN {X 0,Y 443.224,Z 943.906,A -85,B 0,C 180,E1 21668.15,E2 21668.15} C_VEL
LIN {X 0,Y 444.92,Z 931.477,A -85,B 0,C 180,E1 21665.436,E2 21665.436} C_VEL
LIN {X 0,Y 447.388,Z 915.414,A -85,B 0,C 180,E1 21662.447,E2 21662.447} C_VEL
LIN {X 0,Y 449.942,Z 900.024,A -85,B 0,C 180,E1 21660.004,E2 21660.004} C_VEL
LIN {X 0,Y 452.841,Z 883.34,A -85,B 0,C 180,E1 21657.705,E2 21657.705} C_VEL
LIN {X 0,Y 455.647,Z 866.947,A -85,B 0,C 180,E1 21655.765,E2 21655.765} C_VEL
LIN {X 0,Y 458.845,Z 847.836,A -85,B 0,C 180,E1 21653.81,E2 21653.81} C_VEL
LIN {X 0,Y 461.792,Z 829.487,A -85,B 0,C 180,E1 21652.213,E2 21652.213} C_VEL
LIN {X 0,Y 464.82,Z 808.957,A -85,B 0,C 180,E1 21650.697,E2 21650.697} C_VEL
LIN {X 0,Y 467.352,Z 789.911,A -85,B 0,C 180,E1 21649.515,E2 21649.515} C_VEL
LIN {X 0,Y 469.935,Z 767.403,A -85,B 0,C 180,E1 21648.372,E2 21648.372} C_VEL
LIN {X 0,Y 472.103,Z 745.265,A -85,B 0,C 180,E1 21647.486,E2 21647.486} C_VEL
LIN {X 0,Y 473.7,Z 723.281,A -85,B 0,C 180,E1 21646.832,E2 21646.832} C_VEL
LIN {X 0,Y 474.843,Z 700.216,A -85,B 0,C 180,E1 21646.339,E2 21646.339} C_VEL
LIN {X 0,Y 480.957,Z 490.417,A -85,B 0,C 180,E1 21642.666,E2 21642.666} C_VEL
LIN {X 0,Y 482.647,Z 432.418,A -85,B 0,C 180,E1 21641.622,E2 21641.622} C_VEL
LIN {X 0,Y 469.606,Z 413.809,A -85,B 0,C 180,E1 21639.343,E2 21639.343} C_VEL
LIN {X 0,Y 461.353,Z 402.878,A -85,B 0,C 180,E1 21637.791,E2 21637.791} C_VEL
LIN {X 0,Y 457.601,Z 397.974,A -85,B 0,C 180,E1 21637.05,E2 21637.05} C_VEL
LIN {X 0,Y 453.913,Z 393.214,A -85,B 0,C 180,E1 21636.299,E2 21636.299} C_VEL
LIN {X 0,Y 450.679,Z 389.043,A -85,B 0,C 180,E1 21635.618,E2 21635.618} C_VEL
LIN {X 0,Y 449.521,Z 387.633,A -85,B 0,C 180,E1 21635.371,E2 21635.371} C_VEL
LIN {X 0,Y 446.586,Z 384.185,A -85,B 0,C 180,E1 21634.736,E2 21634.736} C_VEL
LIN {X 0,Y 445.381,Z 382.143,A -85,B 0,C 180,E1 21634.453,E2 21634.453} C_VEL
LIN {X 0,Y 442.568,Z 379.633,A -85,B 0,C 180,E1 21633.842,E2 21633.842} C_VEL
LIN {X 0,Y 441.281,Z 376.637,A -85,B 0,C 180,E1 21633.502,E2 21633.502} C_VEL
LIN {X 0,Y 441.185,Z 376.059,A -85,B 0,C 180,E1 21633.459,E2 21633.459} C_VEL
LIN {X 0,Y 441.2,Z 376.048,A -85,B 0,C 180,E1 21629.756,E2 21629.756} C_VEL
LIN {X 0,Y 441.176,Z 376.094,A -85,B 0,C 180,E1 21626.083,E2 21626.083} C_VEL
LIN {X 0,Y 441.15,Z 376.059,A -85,B 0,C 180,E1 21622.382,E2 21622.382} C_VEL
LIN {X 0,Y 441.149,Z 376.067,A -85,B 0,C 180,E1 21618.637,E2 21618.637} C_VEL
LIN {X 0,Y 441.17,Z 376.075,A -85,B 0,C 180,E1 21614.973,E2 21614.973} C_VEL
LIN {X 0,Y 441.189,Z 376.082,A -85,B 0,C 180,E1 21611.239,E2 21611.239} C_VEL
LIN {X 0,Y 441.159,Z 376.086,A -85,B 0,C 180,E1 21607.554,E2 21607.554} C_VEL
LIN {X 0,Y 441.132,Z 376.093,A -85,B 0,C 180,E1 21603.899,E2 21603.899} C_VEL
LIN {X 0,Y 441.128,Z 376.095,A -85,B 0,C 180,E1 21600.13,E2 21600.13} C_VEL
LIN {X 0,Y 441.149,Z 376.091,A -85,B 0,C 180,E1 21596.492,E2 21596.492} C_VEL
LIN {X 0,Y 441.18,Z 376.088,A -85,B 0,C 180,E1 21592.709,E2 21592.709} C_VEL
LIN {X 0,Y 441.156,Z 376.095,A -85,B 0,C 180,E1 21588.892,E2 21588.892} C_VEL
LIN {X 0,Y 441.126,Z 376.1,A -85,B 0,C 180,E1 21585.294,E2 21585.294} C_VEL
LIN {X 0,Y 441.124,Z 376.059,A -85,B 0,C 180,E1 21581.499,E2 21581.499} C_VEL
LIN {X 0,Y 441.152,Z 376.078,A -85,B 0,C 180,E1 21577.9,E2 21577.9} C_VEL
LIN {X 0,Y 441.186,Z 376.083,A -85,B 0,C 180,E1 21574.207,E2 21574.207} C_VEL
LIN {X 0,Y 441.167,Z 376.055,A -85,B 0,C 180,E1 21570.482,E2 21570.482} C_VEL
LIN {X 0,Y 441.212,Z 376.272,A -85,B 0,C 180,E1 21567.907,E2 21567.907} C_VEL
LIN {X 0,Y 442.286,Z 379.301,A -85,B 0,C 180,E1 21567.297,E2 21567.297} C_VEL
LIN {X 0,Y 443.994,Z 381.727,A -85,B 0,C 180,E1 21566.656,E2 21566.656} C_VEL
LIN {X 0,Y 446.206,Z 385.676,A -85,B 0,C 180,E1 21565.776,E2 21565.776} C_VEL
LIN {X 0,Y 449.972,Z 390.853,A -85,B 0,C 180,E1 21564.943,E2 21564.943} C_VEL
LIN {X 0,Y 461.49,Z 406.654,A -85,B 0,C 180,E1 21562.575,E2 21562.575} C_VEL
LIN {X 0,Y 473.772,Z 424.836,A -85,B 0,C 180,E1 21560.269,E2 21560.269} C_VEL
LIN {X 0,Y 482.935,Z 439.57,A -85,B 0,C 180,E1 21558.665,E2 21558.665} C_VEL
LIN {X 0,Y 476.705,Z 650.161,A -85,B 0,C 180,E1 21554.959,E2 21554.959} C_VEL
LIN {X 0,Y 474.051,Z 739.119,A -85,B 0,C 180,E1 21553.39,E2 21553.39} C_VEL
LIN {X 0,Y 472.444,Z 762.41,A -85,B 0,C 180,E1 21552.792,E2 21552.792} C_VEL
LIN {X 0,Y 470.53,Z 784.724,A -85,B 0,C 180,E1 21552.012,E2 21552.012} C_VEL
LIN {X 0,Y 468.21,Z 805.863,A -85,B 0,C 180,E1 21551.049,E2 21551.049} C_VEL
LIN {X 0,Y 465.581,Z 827.248,A -85,B 0,C 180,E1 21549.865,E2 21549.865} C_VEL
LIN {X 0,Y 462.692,Z 847.667,A -85,B 0,C 180,E1 21548.484,E2 21548.484} C_VEL
LIN {X 0,Y 459.603,Z 868.518,A -85,B 0,C 180,E1 21546.815,E2 21546.815} C_VEL
LIN {X 0,Y 456.777,Z 886.308,A -85,B 0,C 180,E1 21545.144,E2 21545.144} C_VEL
LIN {X 0,Y 453.561,Z 906.086,A -85,B 0,C 180,E1 21542.987,E2 21542.987} C_VEL
LIN {X 0,Y 450.89,Z 922.668,A -85,B 0,C 180,E1 21540.888,E2 21540.888} C_VEL
LIN {X 0,Y 448.279,Z 938.952,A -85,B 0,C 180,E1 21538.504,E2 21538.504} C_VEL
LIN {X 0,Y 446.215,Z 952.743,A -85,B 0,C 180,E1 21536.192,E2 21536.192} C_VEL
LIN {X 0,Y 444.302,Z 965.814,A -85,B 0,C 180,E1 21533.611,E2 21533.611} C_VEL
LIN {X 0,Y 442.765,Z 977.731,A -85,B 0,C 180,E1 21530.902,E2 21530.902} C_VEL
LIN {X 0,Y 441.597,Z 988.148,A -85,B 0,C 180,E1 21528.069,E2 21528.069} C_VEL
LIN {X 0,Y 440.792,Z 997.289,A -85,B 0,C 180,E1 21525.12,E2 21525.12} C_VEL
LIN {X 0,Y 440.329,Z 1003.957,A -85,B 0,C 180,E1 21522.457,E2 21522.457} C_VEL
LIN {X 0,Y 440.052,Z 1009.81,A -85,B 0,C 180,E1 21519.547,E2 21519.547} C_VEL
LIN {X 0,Y 439.937,Z 1013.8,A -85,B 0,C 180,E1 21516.787,E2 21516.787} C_VEL
LIN {X 0,Y 439.909,Z 1016.632,A -85,B 0,C 180,E1 21513.91,E2 21513.91} C_VEL
LIN {X 0,Y 439.894,Z 1017.826,A -85,B 0,C 180,E1 21511.042,E2 21511.042} C_VEL
LIN {X 0,Y 439.907,Z 1017.735,A -85,B 0,C 180,E1 21508.438,E2 21508.438} C_VEL
LIN {X 0,Y 439.908,Z 1016.069,A -85,B 0,C 180,E1 21505.438,E2 21505.438} C_VEL
LIN {X 0,Y 439.935,Z 1013.321,A -85,B 0,C 180,E1 21502.82,E2 21502.82} C_VEL
LIN {X 0,Y 440.085,Z 1008.593,A -85,B 0,C 180,E1 21499.794,E2 21499.794} C_VEL
LIN {X 0,Y 440.386,Z 1003.048,A -85,B 0,C 180,E1 21497.146,E2 21497.146} C_VEL
LIN {X 0,Y 440.989,Z 994.768,A -85,B 0,C 180,E1 21494.014,E2 21494.014} C_VEL
LIN {X 0,Y 441.842,Z 985.86,A -85,B 0,C 180,E1 21491.259,E2 21491.259} C_VEL
LIN {X 0,Y 443.128,Z 974.671,A -85,B 0,C 180,E1 21488.375,E2 21488.375} C_VEL
LIN {X 0,Y 444.762,Z 962.641,A -85,B 0,C 180,E1 21485.711,E2 21485.711} C_VEL
LIN {X 0,Y 446.667,Z 949.639,A -85,B 0,C 180,E1 21483.264,E2 21483.264} C_VEL
LIN {X 0,Y 449.012,Z 934.492,A -85,B 0,C 180,E1 21480.797,E2 21480.797} C_VEL
LIN {X 0,Y 451.661,Z 917.741,A -85,B 0,C 180,E1 21478.461,E2 21478.461} C_VEL
LIN {X 0,Y 454.724,Z 899.035,A -85,B 0,C 180,E1 21476.204,E2 21476.204} C_VEL
LIN {X 0,Y 457.54,Z 881.538,A -85,B 0,C 180,E1 21474.382,E2 21474.382} C_VEL
LIN {X 0,Y 460.674,Z 861.348,A -85,B 0,C 180,E1 21472.581,E2 21472.581} C_VEL
LIN {X 0,Y 463.517,Z 842.229,A -85,B 0,C 180,E1 21471.124,E2 21471.124} C_VEL
LIN {X 0,Y 466.28,Z 821.64,A -85,B 0,C 180,E1 21469.807,E2 21469.807} C_VEL
LIN {X 0,Y 468.642,Z 802.129,A -85,B 0,C 180,E1 21468.763,E2 21468.763} C_VEL
LIN {X 0,Y 471.032,Z 778.781,A -85,B 0,C 180,E1 21467.762,E2 21467.762} C_VEL
LIN {X 0,Y 472.987,Z 756.078,A -85,B 0,C 180,E1 21467.019,E2 21467.019} C_VEL
LIN {X 0,Y 474.313,Z 732.908,A -85,B 0,C 180,E1 21466.49,E2 21466.49} C_VEL
LIN {X 0,Y 480.222,Z 528.135,A -85,B 0,C 180,E1 21462.903,E2 21462.903} C_VEL
LIN {X 0,Y 482.788,Z 439.179,A -85,B 0,C 180,E1 21461.31,E2 21461.31} C_VEL
LIN {X 0,Y 472.283,Z 422.593,A -85,B 0,C 180,E1 21459.468,E2 21459.468} C_VEL
LIN {X 0,Y 460.792,Z 405.664,A -85,B 0,C 180,E1 21457.296,E2 21457.296} C_VEL
LIN {X 0,Y 449.801,Z 390.684,A -85,B 0,C 180,E1 21455.033,E2 21455.033} C_VEL
LIN {X 0,Y 445.732,Z 385.136,A -85,B 0,C 180,E1 21454.11,E2 21454.11} C_VEL
LIN {X 0,Y 443.683,Z 380.978,A -85,B 0,C 180,E1 21453.203,E2 21453.203} C_VEL
LIN {X 0,Y 441.576,Z 377.804,A -85,B 0,C 180,E1 21452.384,E2 21452.384} C_VEL
LIN {X 0,Y 441.192,Z 376.089,A -85,B 0,C 180,E1 21452.026,E2 21452.026} C_VEL
LIN {X 0,Y 441.148,Z 376.057,A -85,B 0,C 180,E1 21448.422,E2 21448.422} C_VEL
LIN {X 0,Y 441.132,Z 376.06,A -85,B 0,C 180,E1 21444.791,E2 21444.791} C_VEL
LIN {X 0,Y 441.151,Z 376.091,A -85,B 0,C 180,E1 21441.123,E2 21441.123} C_VEL
LIN {X 0,Y 441.172,Z 376.044,A -85,B 0,C 180,E1 21437.407,E2 21437.407} C_VEL
LIN {X 0,Y 441.153,Z 376.097,A -85,B 0,C 180,E1 21433.767,E2 21433.767} C_VEL
LIN {X 0,Y 441.121,Z 376.098,A -85,B 0,C 180,E1 21430.183,E2 21430.183} C_VEL
LIN {X 0,Y 441.116,Z 376.095,A -85,B 0,C 180,E1 21426.376,E2 21426.376} C_VEL
LIN {X 0,Y 441.143,Z 376.088,A -85,B 0,C 180,E1 21422.728,E2 21422.728} C_VEL
LIN {X 0,Y 441.18,Z 376.084,A -85,B 0,C 180,E1 21419.091,E2 21419.091} C_VEL
LIN {X 0,Y 441.151,Z 376.088,A -85,B 0,C 180,E1 21415.32,E2 21415.32} C_VEL
LIN {X 0,Y 441.13,Z 376.091,A -85,B 0,C 180,E1 21411.79,E2 21411.79} C_VEL
LIN {X 0,Y 441.145,Z 376.086,A -85,B 0,C 180,E1 21408.097,E2 21408.097} C_VEL
LIN {X 0,Y 441.188,Z 376.074,A -85,B 0,C 180,E1 21404.489,E2 21404.489} C_VEL
LIN {X 0,Y 441.185,Z 376.07,A -85,B 0,C 180,E1 21400.678,E2 21400.678} C_VEL
LIN {X 0,Y 441.154,Z 376.056,A -85,B 0,C 180,E1 21397.056,E2 21397.056} C_VEL
LIN {X 0,Y 441.152,Z 376.096,A -85,B 0,C 180,E1 21393.336,E2 21393.336} C_VEL
LIN {X 0,Y 441.164,Z 376.056,A -85,B 0,C 180,E1 21389.641,E2 21389.641} C_VEL
LIN {X 0,Y 441.204,Z 376.196,A -85,B 0,C 180,E1 21386.42,E2 21386.42} C_VEL
LIN {X 0,Y 442.248,Z 379.137,A -85,B 0,C 180,E1 21386.13,E2 21386.13} C_VEL
LIN {X 0,Y 444.764,Z 381.786,A -85,B 0,C 180,E1 21385.571,E2 21385.571} C_VEL
LIN {X 0,Y 445.862,Z 382.76,A -85,B 0,C 180,E1 21385.336,E2 21385.336} C_VEL
LIN {X 0,Y 448.26,Z 386.461,A -85,B 0,C 180,E1 21384.789,E2 21384.789} C_VEL
LIN {X 0,Y 450.482,Z 388.707,A -85,B 0,C 180,E1 21384.325,E2 21384.325} C_VEL
LIN {X 0,Y 453.569,Z 392.893,A -85,B 0,C 180,E1 21383.669,E2 21383.669} C_VEL
LIN {X 0,Y 455.352,Z 395.027,A -85,B 0,C 180,E1 21383.307,E2 21383.307} C_VEL
LIN {X 0,Y 464.01,Z 406.366,A -85,B 0,C 180,E1 21381.601,E2 21381.601} C_VEL
LIN {X 0,Y 474.254,Z 420.383,A -85,B 0,C 180,E1 21379.725,E2 21379.725} C_VEL
LIN {X 0,Y 482.723,Z 432.792,A -85,B 0,C 180,E1 21378.267,E2 21378.267} C_VEL
LIN {X 0,Y 476.739,Z 632.848,A -85,B 0,C 180,E1 21374.742,E2 21374.742} C_VEL
LIN {X 0,Y 475.797,Z 666.177,A -85,B 0,C 180,E1 21374.161,E2 21374.161} C_VEL
LIN {X 0,Y 474.899,Z 673.878,A -85,B 0,C 180,E1 21374.111,E2 21374.111} C_VEL
LIN {X 0,Y 469.85,Z 694.47,A -85,B 0,C 180,E1 21374.292,E2 21374.292} C_VEL
LIN {X 0,Y 469.061,Z 701.067,A -85,B 0,C 180,E1 21374.235,E2 21374.235} C_VEL
LIN {X 0,Y 467.871,Z 723.81,A -85,B 0,C 180,E1 21373.742,E2 21373.742} C_VEL
LIN {X 0,Y 466.178,Z 745.937,A -85,B 0,C 180,E1 21373.076,E2 21373.076} C_VEL
LIN {X 0,Y 464.037,Z 766.847,A -85,B 0,C 180,E1 21372.236,E2 21372.236} C_VEL
LIN {X 0,Y 461.392,Z 788.987,A -85,B 0,C 180,E1 21371.118,E2 21371.118} C_VEL
LIN {X 0,Y 458.697,Z 808.262,A -85,B 0,C 180,E1 21369.923,E2 21369.923} C_VEL
LIN {X 0,Y 455.383,Z 829.729,A -85,B 0,C 180,E1 21368.33,E2 21368.33} C_VEL
LIN {X 0,Y 452.282,Z 848.031,A -85,B 0,C 180,E1 21366.721,E2 21366.721} C_VEL
LIN {X 0,Y 448.823,Z 867.466,A -85,B 0,C 180,E1 21364.711,E2 21364.711} C_VEL
LIN {X 0,Y 445.717,Z 884.644,A -85,B 0,C 180,E1 21362.645,E2 21362.645} C_VEL
LIN {X 0,Y 442.71,Z 900.78,A -85,B 0,C 180,E1 21360.374,E2 21360.374} C_VEL
LIN {X 0,Y 439.967,Z 916.24,A -85,B 0,C 180,E1 21357.867,E2 21357.867} C_VEL
LIN {X 0,Y 437.761,Z 929.134,A -85,B 0,C 180,E1 21355.426,E2 21355.426} C_VEL
LIN {X 0,Y 435.644,Z 942.971,A -85,B 0,C 180,E1 21352.392,E2 21352.392} C_VEL
LIN {X 0,Y 434.251,Z 953.769,A -85,B 0,C 180,E1 21349.641,E2 21349.641} C_VEL
LIN {X 0,Y 433.204,Z 963.417,A -85,B 0,C 180,E1 21346.696,E2 21346.696} C_VEL
LIN {X 0,Y 432.56,Z 971.146,A -85,B 0,C 180,E1 21343.873,E2 21343.873} C_VEL
LIN {X 0,Y 432.173,Z 977.491,A -85,B 0,C 180,E1 21340.934,E2 21340.934} C_VEL
LIN {X 0,Y 432,Z 982.427,A -85,B 0,C 180,E1 21337.981,E2 21337.981} C_VEL
LIN {X 0,Y 431.918,Z 985.689,A -85,B 0,C 180,E1 21335.046,E2 21335.046} C_VEL
LIN {X 0,Y 431.909,Z 987.437,A -85,B 0,C 180,E1 21332.388,E2 21332.388} C_VEL
LIN {X 0,Y 431.884,Z 987.901,A -85,B 0,C 180,E1 21329.336,E2 21329.336} C_VEL
LIN {X 0,Y 431.886,Z 987.075,A -85,B 0,C 180,E1 21326.815,E2 21326.815} C_VEL
LIN {X 0,Y 431.934,Z 984.811,A -85,B 0,C 180,E1 21323.888,E2 21323.888} C_VEL
LIN {X 0,Y 432.027,Z 981.119,A -85,B 0,C 180,E1 21321.08,E2 21321.08} C_VEL
LIN {X 0,Y 432.263,Z 975.781,A -85,B 0,C 180,E1 21318.079,E2 21318.079} C_VEL
LIN {X 0,Y 432.736,Z 968.817,A -85,B 0,C 180,E1 21315.141,E2 21315.141} C_VEL
LIN {X 0,Y 433.555,Z 960.13,A -85,B 0,C 180,E1 21312.14,E2 21312.14} C_VEL
LIN {X 0,Y 434.659,Z 950.488,A -85,B 0,C 180,E1 21309.395,E2 21309.395} C_VEL
LIN {X 0,Y 436.384,Z 937.934,A -85,B 0,C 180,E1 21306.364,E2 21306.364} C_VEL
LIN {X 0,Y 438.392,Z 925.433,A -85,B 0,C 180,E1 21303.742,E2 21303.742} C_VEL
LIN {X 0,Y 440.907,Z 910.78,A -85,B 0,C 180,E1 21301.12,E2 21301.12} C_VEL
LIN {X 0,Y 443.767,Z 895.271,A -85,B 0,C 180,E1 21298.715,E2 21298.715} C_VEL
LIN {X 0,Y 446.766,Z 878.706,A -85,B 0,C 180,E1 21296.521,E2 21296.521} C_VEL
LIN {X 0,Y 450.201,Z 859.904,A -85,B 0,C 180,E1 21294.376,E2 21294.376} C_VEL
LIN {X 0,Y 453.156,Z 843.047,A -85,B 0,C 180,E1 21292.728,E2 21292.728} C_VEL
LIN {X 0,Y 456.556,Z 822.266,A -85,B 0,C 180,E1 21290.991,E2 21290.991} C_VEL
LIN {X 0,Y 459.439,Z 803.172,A -85,B 0,C 180,E1 21289.648,E2 21289.648} C_VEL
LIN {X 0,Y 462.311,Z 781.761,A -85,B 0,C 180,E1 21288.403,E2 21288.403} C_VEL
LIN {X 0,Y 464.622,Z 761.804,A -85,B 0,C 180,E1 21287.454,E2 21287.454} C_VEL
LIN {X 0,Y 466.761,Z 738.844,A -85,B 0,C 180,E1 21286.601,E2 21286.601} C_VEL
LIN {X 0,Y 468.193,Z 719.021,A -85,B 0,C 180,E1 21286.048,E2 21286.048} C_VEL
LIN {X 0,Y 469.467,Z 687.537,A -85,B 0,C 180,E1 21285.438,E2 21285.438} C_VEL
LIN {X 0,Y 476.06,Z 475.787,A -85,B 0,C 180,E1 21281.692,E2 21281.692} C_VEL
LIN {X 0,Y 477.193,Z 436.369,A -85,B 0,C 180,E1 21280.963,E2 21280.963} C_VEL
LIN {X 0,Y 465.734,Z 419.861,A -85,B 0,C 180,E1 21278.899,E2 21278.899} C_VEL
LIN {X 0,Y 457.072,Z 408.283,A -85,B 0,C 180,E1 21277.226,E2 21277.226} C_VEL
LIN {X 0,Y 450.62,Z 399.842,A -85,B 0,C 180,E1 21275.897,E2 21275.897} C_VEL
LIN {X 0,Y 446.144,Z 394.204,A -85,B 0,C 180,E1 21274.932,E2 21274.932} C_VEL
LIN {X 0,Y 442.966,Z 390.074,A -85,B 0,C 180,E1 21274.217,E2 21274.217} C_VEL
LIN {X 0,Y 441.78,Z 388.732,A -85,B 0,C 180,E1 21273.949,E2 21273.949} C_VEL
LIN {X 0,Y 438.845,Z 385.298,A -85,B 0,C 180,E1 21273.27,E2 21273.27} C_VEL
LIN {X 0,Y 437.811,Z 383.335,A -85,B 0,C 180,E1 21273.003,E2 21273.003} C_VEL
LIN {X 0,Y 434.956,Z 381.12,A -85,B 0,C 180,E1 21272.347,E2 21272.347} C_VEL
LIN {X 0,Y 433.473,Z 378.171,A -85,B 0,C 180,E1 21271.942,E2 21271.942} C_VEL
LIN {X 0,Y 433.262,Z 377.081,A -85,B 0,C 180,E1 21271.845,E2 21271.845} C_VEL
LIN {X 0,Y 433.241,Z 377.048,A -85,B 0,C 180,E1 21268.087,E2 21268.087} C_VEL
LIN {X 0,Y 433.213,Z 377.043,A -85,B 0,C 180,E1 21264.402,E2 21264.402} C_VEL
LIN {X 0,Y 433.216,Z 377.086,A -85,B 0,C 180,E1 21260.679,E2 21260.679} C_VEL
LIN {X 0,Y 433.23,Z 377.03,A -85,B 0,C 180,E1 21257.044,E2 21257.044} C_VEL
LIN {X 0,Y 433.256,Z 377.081,A -85,B 0,C 180,E1 21253.343,E2 21253.343} C_VEL
LIN {X 0,Y 433.226,Z 377.083,A -85,B 0,C 180,E1 21249.566,E2 21249.566} C_VEL
LIN {X 0,Y 433.197,Z 377.085,A -85,B 0,C 180,E1 21245.913,E2 21245.913} C_VEL
LIN {X 0,Y 433.191,Z 377.083,A -85,B 0,C 180,E1 21242.117,E2 21242.117} C_VEL
LIN {X 0,Y 433.203,Z 377.079,A -85,B 0,C 180,E1 21238.413,E2 21238.413} C_VEL
LIN {X 0,Y 433.23,Z 377.073,A -85,B 0,C 180,E1 21234.703,E2 21234.703} C_VEL
LIN {X 0,Y 433.21,Z 377.076,A -85,B 0,C 180,E1 21230.971,E2 21230.971} C_VEL
LIN {X 0,Y 433.185,Z 377.078,A -85,B 0,C 180,E1 21227.334,E2 21227.334} C_VEL
LIN {X 0,Y 433.183,Z 377.058,A -85,B 0,C 180,E1 21223.645,E2 21223.645} C_VEL
LIN {X 0,Y 433.209,Z 377.078,A -85,B 0,C 180,E1 21219.929,E2 21219.929} C_VEL
LIN {X 0,Y 433.245,Z 377.038,A -85,B 0,C 180,E1 21216.324,E2 21216.324} C_VEL
LIN {X 0,Y 433.23,Z 377.064,A -85,B 0,C 180,E1 21212.511,E2 21212.511} C_VEL
LIN {X 0,Y 433.213,Z 377.089,A -85,B 0,C 180,E1 21209.441,E2 21209.441} C_VEL
LIN {X 0,Y 434.24,Z 380.122,A -85,B 0,C 180,E1 21208.797,E2 21208.797} C_VEL
LIN {X 0,Y 435.965,Z 382.145,A -85,B 0,C 180,E1 21208.164,E2 21208.164} C_VEL
LIN {X 0,Y 437.379,Z 385.411,A -85,B 0,C 180,E1 21207.506,E2 21207.506} C_VEL
LIN {X 0,Y 440.043,Z 388.662,A -85,B 0,C 180,E1 21206.876,E2 21206.876} C_VEL
LIN {X 0,Y 443.967,Z 393.823,A -85,B 0,C 180,E1 21205.969,E2 21205.969} C_VEL
LIN {X 0,Y 448.989,Z 400.645,A -85,B 0,C 180,E1 21204.855,E2 21204.855} C_VEL
LIN {X 0,Y 458.038,Z 413.182,A -85,B 0,C 180,E1 21202.972,E2 21202.972} C_VEL
LIN {X 0,Y 469.778,Z 430.716,A -85,B 0,C 180,E1 21200.715,E2 21200.715} C_VEL
LIN {X 0,Y 477.516,Z 443.341,A -85,B 0,C 180,E1 21199.318,E2 21199.318} C_VEL
LIN {X 0,Y 470.959,Z 652.683,A -85,B 0,C 180,E1 21195.601,E2 21195.601} C_VEL
LIN {X 0,Y 468.231,Z 738.936,A -85,B 0,C 180,E1 21194.064,E2 21194.064} C_VEL
LIN {X 0,Y 466.533,Z 762.244,A -85,B 0,C 180,E1 21193.463,E2 21193.463} C_VEL
LIN {X 0,Y 464.441,Z 785.182,A -85,B 0,C 180,E1 21192.651,E2 21192.651} C_VEL
